DATA_BLOCK "dbtags_Sterowanie"   // DB1
{ S7_Optimized_Access := 'FALSE' }
VERSION : 0.1
// stored: AutoNumber false, DBAccessibleFromOPCUA true, IsOnlyStoredInLoadMemory false, IsWriteProtectedInAS false
   VAR RETAIN
      PID_Compact : Struct
         Setpoint : Real := 1.5;
         Input : Real;
         Input_PER : Int;
         Disturbance : Real;
         ManualEnable : Bool;
         ManualValue : Real;
         ErrorAck : Bool;
         Reset : Bool;
         ModeActivate : Bool;
         Mode : Int := 3;
         ScaledInput : Real;
         Output : Real;
         Output_PER : Int;
         Output_PWM : Bool;
         SetpointLimit_H : Bool;
         SetpointLimit_L : Bool;
         InputWarning_H : Bool;
         InputWarning_L : Bool;
         State : Int;
         Error : Bool;
         ErrorBits : DWord;
      END_STRUCT;
      Tuning : Struct
         Mode : Int := 1;
         Mode_visible : Bool;
         SUT_visible : Bool;
         TIR_visible : Bool;
         last_state : Int;
      END_STRUCT;
      HMI : Struct
         PhysicalUnit : String[5] := '1/min';
         Output_PWM_USInt : USInt;
         "position reached" : Bool;
         ManualMode_visible : Bool;
         Setpoint_limited : Bool;
         ErrorBits_Int : Int;
         ErrorAck_Int : Int;
         Warning_Int : Int;
         ErrorAck_Int_edge : Bool;   // pamięć zbocza reset PID po error
         ErrorAck : Bool;   // reset błędu PID
         Acknowledge_visible : Bool;
      END_STRUCT;
      Speed : Struct
         encoder : Real;
         rpm : Real;
      END_STRUCT;
      SetupControlPompownia : Struct
         SV : Real := 2.0;
         r_Pv_Norm_OUT_2 : Real := 10.0;   // Zakres górny wejścia In_PER_PID
         r_Pv_Norm_OUT_1 : Real := 0.0;   // Zakres dolny wejścia In_PER_PID
         r_Lmn_Hlm : Real := 100.0;   // Ograniczenie górne wartości procesowej [%] MV
         r_Lmn_Llm : Real := 0.0;   // Ograniczenie dolne wartości procesowej [%] MV
         r_Sp_Hlm : Real := 8.0;   // Ograniczenie H zakresu zadawania wartości ciśnienie SV
         r_Sp_Llm : Real := 0.0;   // Ograniczenie L zakresu zadawania wartości ciśnienia SV
         r_Pv_HWrn : Real := 7.8;   // Ostrzeżenie wysoki dla PV
         r_Pv_LWrn : Real := 5.3;   // Ostrzeżenie niski dla PV
         r_Pv_Hlm : Real := 10.0;   // Przetwornik Limit górny
         r_Pv_Llm : Real := 0.0;   // Przetwornik Limit dlolny
         Time_ONK1 : Int := 90;
         Time_ONK2 : Int := 90;
         Time_OFFK1 : Int := 5;
         Time_OFFK2 : Int := 5;
         TimeHz : Int := 30;
         NO4_Cureent : Real;   // Aktualna zawartość amoniaku
         CureentValue_O2_1 : Real;   // Przyrost ciśnienia 1
         CureentValue_O2_2 : Real;   // Przyrost ciścienia 2
         Data_sek1 : Int;   // Licznik sekund dla pomiaru nr1 funkcji Calculation_of_the_increment
         Data_sek2 : Int;   // Licznik sekund dla pomiaru nr2 funkcji Calculation_of_the_increment
         Static_1 : Word;
         Z11_Status : Word;   // Status napędu copia z SCADA
         Z12_Status : Word;   // Status napędu copia z SCADA
         Static_2 : Real;
         Switch_Aut_Rem_Pompy : Bool;   // Bit przełacznika trybu pracy pomp
         tagsdbSwitch_ModelSterowania : Word;   // Wybur model sterowania0- wyłączone, 1- Dosilanie, 2- Przetłączanie, 3- Automat, 4- Ręczne
         barMax_Manual_Hz : Real := 5.0;   // Instancja wartości zadawanej w trybie manual do regulatora PID gdy ciśnienie w rurociągu max
         CurrentMax_Manual_Hz : Real := 5.0;   // Instancja wartości zadawanej w trybie manual do regulatora PID gdy przeciążony falownik
         Statut_Motor : Byte;   // Byte stanu gotowości pomp
         Mem_Res_setCMD_MC_P1 : Bool;   // Znacznik 50 Hz podtrzymanie przełączenia na sieć
         Mem_Res_setCMD_MC_P2 : Bool;   // Znacznik 50 Hz podtrzymanie przełączenia na sieć
         Mem_Res_setCMD_MC_P3 : Bool;   // Znacznik 50 Hz podtrzymanie przełączenia na sieć
         Switch_In_Analog_Mudbas : Bool;   // Bit przełączeania pomiędzy sygnałem bar z wej analog / Modbus
         PV_HWrn_correction : Real;   // Wspóczninik służący wprowadzeniu korekty ostrzeżenia przekroczenia wartości zadanej ciśnienie
         PV_LWrn_correction : Real;   // Wspóczninik służący wprowadzeniu korekty ostrzeżenia zbyt niskia wartości ciśnieniea w stosunku do zadanej
         TimerSet_O2_Up : IEC_TIMER;   // Czas opóżninia podniesienia zadanej wartości ciśnienia
         TimerSet_O2_Down : IEC_TIMER;   // Czas opóżninia obniżenia zadanej wartości ciśnienia
         Pv_Llm_B8 : Real := -1.0;   // Limit dolny przetwornika ciśnienie B8
         Pv_Hlm_B8 : Real := 2.0;   // Limit górny przetwornika ciśnienia B8
         Time_ONK3 : Int;
         Time_OFFK3 : Int := 0;
         Setpoint_Inverter_Pompy { ExternalAccessible := 'False'; ExternalVisible := 'False'; ExternalWritable := 'False'} : Real;   // Wartość zadana Hz odczytane z Modbus
         Frequency_inverter_Pompy { ExternalAccessible := 'False'; ExternalVisible := 'False'; ExternalWritable := 'False'} : Real;   // Aktualne Hz silniku odczytane z Modbus
         MotorCurrent_Inverter_Pompy { ExternalAccessible := 'False'; ExternalVisible := 'False'; ExternalWritable := 'False'} : Real;   // Prąd na silniku zasilanym z falownika odczytane z Modbus
         NormalCurrent_InverterPompy { ExternalAccessible := 'False'; ExternalVisible := 'False'; ExternalWritable := 'False'} : Real;   // Prąd nominalny falownika odczytane z Modbus
         MaxCurrent_Inverter_Pompy { ExternalAccessible := 'False'; ExternalVisible := 'False'; ExternalWritable := 'False'} : Real;   // Prad Max krótkotrwały odczytane z Modbus
         OverTemp_InverterPompy { ExternalAccessible := 'False'; ExternalVisible := 'False'; ExternalWritable := 'False'} : Word;
         OverVolta_InverterPompy { ExternalAccessible := 'False'; ExternalVisible := 'False'; ExternalWritable := 'False'} : Word;
         PIF_Reset : IEC_TIMER;   // impuls resetu regulatora PID 1
         mbAdresABB_Q1 : Word := 1;   // Adres modbus przepływomierz pompownia
         mbAdresPompy : Word := 26;   // Adres modbus falownik
         mbAdresrezerwa_Q2 : Word;   // Adres modbus przepływomierz magistrala - w Stacji Zasuw
         mbAdres_IDslave : Word := 2;   // Adres modbus MT101
         SubPV_K1 : Real := 0.6;   // Wspólczynnik pomniejszenia wyliczanego ciśnienia napotrzeby wyłączenia dodatowej pompy
         SubPV_K2 : Real := 0.45;   // Wspólczynnik pomniejszenia wyliczanego ciśnieia napotrzeby wyłączenia dodatowej pompy
         Setpoint_Inverter_a { ExternalAccessible := 'False'; ExternalVisible := 'False'; ExternalWritable := 'False'} : Real;   // Wartość zadana Hz odczytane z Modbus
         Frequency_inverter_a { ExternalAccessible := 'False'; ExternalVisible := 'False'; ExternalWritable := 'False'} : Real;   // Aktualne Hz silniku odczytane z Modbus
         MotorCurrent_Inverter_a { ExternalAccessible := 'False'; ExternalVisible := 'False'; ExternalWritable := 'False'} : Real;   // Prąd na silniku zasilanym z falownika odczytane z Modbus
         NormalCurrent_Inverter_a { ExternalAccessible := 'False'; ExternalVisible := 'False'; ExternalWritable := 'False'} : Real;   // Prąd nominalny falownika odczytane z Modbus
         MaxCurrent_Inverter_a { ExternalAccessible := 'False'; ExternalVisible := 'False'; ExternalWritable := 'False'} : Real;   // Prad Max krótkotrwały odczytane z Modbus
         OverTemp_InverterPomp { ExternalAccessible := 'False'; ExternalVisible := 'False'; ExternalWritable := 'False'} : Word;
         OverVolta_InverterPomp { ExternalAccessible := 'False'; ExternalVisible := 'False'; ExternalWritable := 'False'} : Word;
         set_barDN500_B5 { ExternalAccessible := 'False'; ExternalVisible := 'False'; ExternalWritable := 'False'} : Real;   // Zadane ciśnienie dosilanie DN500 na czujniku B5
         set_barDN225_B6 { ExternalAccessible := 'False'; ExternalVisible := 'False'; ExternalWritable := 'False'} : Real;   // Zadane ciśnienie przetłacania DN225 na czujniku B6
         MotorCurrent_Inverter_b { ExternalAccessible := 'False'; ExternalVisible := 'False'; ExternalWritable := 'False'} : Real;   // Prąd na silniku zasilanym z falownika odczytane z Modbus
         NormalCurrent_Inverter_b { ExternalAccessible := 'False'; ExternalVisible := 'False'; ExternalWritable := 'False'} : Real;   // Prąd nominalny falownika odczytane z Modbus
         MaxCurrent_Inverter_b { ExternalAccessible := 'False'; ExternalVisible := 'False'; ExternalWritable := 'False'} : Real;   // Prad Max krótkotrwały odczytane z Modbus
         OverTemp_Inverter_b { ExternalAccessible := 'False'; ExternalVisible := 'False'; ExternalWritable := 'False'} : Word;
         OverVolta_Inverter_b { ExternalAccessible := 'False'; ExternalVisible := 'False'; ExternalWritable := 'False'} : Word;
         actOverCurrent_set : Real;   // Zakres ograniczenia prądowego.
         actOverCurrent_set_a : Real := 0.0;   // Zakres ograniczenia prądowego.
         actOverCurrent_set_b : Real := 0.0;   // Zakres ograniczenia prądowego.
         AnalogFrequency_inverter_a { ExternalAccessible := 'False'; ExternalVisible := 'False'; ExternalWritable := 'False'} : Real;   // Aktualne Hz silniku odczytane z Analog
         AnalogFrequency_inverter_b { ExternalAccessible := 'False'; ExternalVisible := 'False'; ExternalWritable := 'False'} : Real := 0.0;   // Aktualne Hz silniku odczytane z Analog
         MaxHour_InverterBlowerWork : Word := 43200;   // Maksymalny czas pracy pracy ciągłej na falowniku dla kompresorów 43200sek = 12h
         TimerSet_Hz_Up_a : IEC_TIMER;
         TimerSet_Hz_Down_a : IEC_TIMER;
         TimerSet_Hz_Up_b : IEC_TIMER;
         TimerSet_Hz_Down_b : IEC_TIMER;
         TimerGen_Hz_Up_a : IEC_TIMER;
         TimerGen_Hz_Down_a : IEC_TIMER;
         TimerGen_Hz_Up_b : IEC_TIMER;
         TimerGen_Hz_Down_b : IEC_TIMER;
         Mem_Res_setCMD_MC_P4 : Bool;   // Znacznik 50 Hz podtrzymanie przełączenia na sieć
         "ABB_1Master.mode" : Byte := 0;
         "rez_2Master.mode" : Byte := 0;
         "Fal_2Master.mode_1" : Byte := 0;
         "Slave_2Master.mode_2" : Byte := 2;
      END_STRUCT;
      "Paramaetry _Zbiorniki" : Struct   // parametry sterowania
         set_poziom_napełniania : Real := 400.0;   // wartość zadana poziomu napełniania
         set_poziom_opróżniania : Real := 30.0;   // wartość zadana poziomu opróżniania
         set_bity_sterowania_napęami_1 : Word;   // bity sterowania napędami
         set_bity_sterowania_napęami_2 : Word;   // bity sterowania napędami
         set_bity_tryb_napędów_1 : Word;   // bity sterowania przełączaniem trybów pracy
         set_bity_tryb_napędów_2 : Word;   // bity sterowania przełączaniem trybów pracy
         rez_alarm_napędów : Word;   // bity kasowania alarmów napędów
         set_strategia_sterowania : Word := 16#0003;   // Sygnały sterowania strategią pompownia - 0= wyłaczone, 1=dosilanie, 2=przetłaczanie,3=automat, 4=ręczne
         set_sterowanie_cyklem : Word;   // Sygnały sterowania cyklem zbiorniki 0-wyłączone, 1=dobowy, 2=tygodniowy, 3=ręczne
         set_położenie_Z10 : Word;   // zadane położenie procentowe Z10
      END_STRUCT;
      Zbiorniki_Godziny : Struct   // godziny cykli pracy
         start_napełnianie : DTL := DTL#1970-01-01-23:55:00;
         Stop_napełnianie : DTL := DTL#1970-01-01-16:00:00;
         Start_przetłaczanie_1 : DTL := DTL#1970-01-01-18:00:00;
         Stop_przetłaczanie_1 : DTL := DTL#1970-01-01-23:55:00;
         Start_dosilanie_1 : DTL := DTL#1970-01-01-18:00:00;
         Stop_dosilanie_1 : DTL := DTL#1970-01-01-23:55:00;
      END_STRUCT;
      Zbiorniki_sondy : Struct   // parametry sond
         "Pv.LIm_Tank1" : Int := 0;   // zakres pomiarowy dolny
         "Pv.HIm_Tank1" : Int := 400;   // zakres pomiarowy górny
         "Pv.LIm_Tank2" : Int := 0;   // zakres pomiarowy dolny
         "Pv.HIm_Tank2" : Int := 400;   // zakres pomiarowy górny
         "Pv.LIm_Tank3" : Int := 0;   // zakres pomiarowy dolny
         "Pv.HIm_Tank3" : Int := 400;   // zakres pomiarowy górny
      END_STRUCT;
      suction_r_Pv_Hlm : Real := 2.0;   // Przetwornik ssania Limit górny
      suction_r_Pv_Llm : Real := -1.0;   // Przetwornik ssania Limit dlolny
   END_VAR
BEGIN
   SetupControlPompownia.PIF_Reset.PT := T#500ms;
   SetupControlPompownia.TimerSet_Hz_Up_a.PT := T#2M;
   SetupControlPompownia.TimerSet_Hz_Down_a.PT := T#2M;
   SetupControlPompownia.TimerSet_Hz_Up_b.PT := T#2M;
   SetupControlPompownia.TimerSet_Hz_Down_b.PT := T#2M;
   SetupControlPompownia.TimerGen_Hz_Up_a.PT := T#100ms;
   SetupControlPompownia.TimerGen_Hz_Down_a.PT := T#100ms;
   SetupControlPompownia.TimerGen_Hz_Up_b.PT := T#100ms;
   SetupControlPompownia.TimerGen_Hz_Down_b.PT := T#100ms;
END_DATA_BLOCK

DATA_BLOCK "hourWork_setData"   // DB30
{ S7_Optimized_Access := 'FALSE' }
VERSION : 0.1
// stored: AutoNumber false, DBAccessibleFromOPCUA true, IsOnlyStoredInLoadMemory false, IsWriteProtectedInAS false
   VAR RETAIN
      Sek_P1 : Int := 1;   // Licznik sekund
      Sek_P2 : Int := 2;   // Licznik sekund
      Sek_P3 : Int := 3;   // Licznik sekund
      Sek_P4 : Int := 3;
      Edge_P1 : Bool;   // Pamięć zbocza
      Edge_P2 : Bool;   // Pamięć zbocza
      Edge_P3 : Bool;   // Pamięć zbocza
      Edge_P4 : Bool := false;
      Sek_a : Int;   // Licznik sekund
      Sek_b : Int;   // Licznik sekund
      Edge_a : Bool;   // Pamięć zbocza
      Edge_b : Bool;   // Pamięć zbocza
      Sum_sek_hur_P1 : Real;   // Licznik sumator godzin i sekund na potrzeby wyznaczania dumchawy do pracy
      Sum_sek_hur_P2 : Real := 0.0;   // Licznik sumator godzin i sekund na potrzeby wyznaczania dumchawy do pracy
      Sum_sek_hur_P3 : Real := 0.0;   // Licznik sumator godzin i sekund na potrzeby wyznaczania dumchawy do pracy
      Sum_sek_hur_P4 : Real := 0.0;
      HourCounterP1 : DWord;   // Counter Work
      HourCounterP2 : DWord;   // Counter Work
      HourCounterP3 : DWord;   // Counter Work
      HourCounterP4 : DWord;
   END_VAR
BEGIN
END_DATA_BLOCK

DATA_BLOCK "dbMasterData"   // DB35
{ S7_Optimized_Access := 'FALSE' }
VERSION : 0.1
// stored: AutoNumber false, DBAccessibleFromOPCUA true, IsOnlyStoredInLoadMemory false, IsWriteProtectedInAS false
   VAR
      ID6_aktualny_przeływu_Adres_33057 { S7_SetPoint := 'True'} : "typeDataABB_real";   // wielkość przepływu / Wartość aktualnego przepływu
      ID6_Licznik_suma_VF_Adres_33063 : "typeDataABB_real";   // licznik objętości VF / Stan licznika objętości dla przepływu w przód VF
      ID6_Licznik_suma_VR_Adres_33065 { S7_SetPoint := 'True'} : "typeDataABB_real";   // licznik objętości VR / Stan licznika objętości dla przepływu w tył VR
      ID6__VD_Adres_6 { S7_SetPoint := 'True'} : "typeDataABB_real";   // Stan bieżącego różnicowego licznika objętości VD
      ID6___GF_Adres_8 { S7_SetPoint := 'True'} : "typeDataABB_real";   // Stan głównego licznika objętości dla przepływu w przód GF
      ID6__GR_Adres_10 { S7_SetPoint := 'True'} : "typeDataABB_real";   // Sta ngłownego licznika objętości dla przepływu w tył GR
      ID6__GD_Adres_12 { S7_SetPoint := 'True'} : "typeDataABB_real";   // Stan głownego licznika różnicowego GD
      ID6__1000 { S7_SetPoint := 'True'} : "typeDataInverter_Word";   // 8-przekrodzony zakres pracy przetwornika, 20-otwarty obwód cewki, 21zwarcie w obwodzie cewki, 26-brak cieczy w czujniku
      data_rez_Wielkość_przeływu_Adres_0 { S7_SetPoint := 'True'} : "typeDataABB_real";   // wielkość przepływu / Wartość aktualnego przepływu
      data_rez_Licznik_objętość_VF_Adres_2 { S7_SetPoint := 'True'} : "typeDataABB_real";   // licznik objętości VF / Stan licznika objętości dla przepływu w przód VF
      data_rez_Licznik_objętość_VR_Adres_4 { S7_SetPoint := 'True'} : "typeDataABB_real";   // licznik objętości VR / Stan licznika objętości dla przepływu w tył VR
      data_rez_Licznik_różnicowy_VD_Adres_6 { S7_SetPoint := 'True'} : "typeDataABB_real";   // licznik różnicy / Stan bieżącego różnicowego licznika objętości VD
      data_rez_Stan_licz_bjętości_GF_Adres_8 { S7_SetPoint := 'True'} : "typeDataABB_real";   // licznik objetosci GF / Stan głównego licznika objętości dla przepływu w przód GF
      data_rez_Stan_licz_bjętości_GR_Adres_10 { S7_SetPoint := 'True'} : "typeDataABB_real";   // licznik objetości GR / Sta ngłownego licznika objętości dla przepływu w tył GR
      data_rez_Stan_licz_rózicowego_obj_GD_Adres_12 { S7_SetPoint := 'True'} : "typeDataABB_real";   // licznik róznicowy / Stan głownego licznika różnicowego GD
      data_rez_Stan_urządzenia_1000 { S7_SetPoint := 'True'} : "typeDataInverter_Word";   // stan urządzenia / 8-przekrodzony zakres pracy przetwornika, 20-otwarty obwód cewki, 21zwarcie w obwodzie cewki, 26-brak cieczy w czujniku
      ID26_Inver_Control_word_416000_Fal { S7_SetPoint := 'True'} : "typeDataInverter_Word";   // Sowo komtrolneCTW falownika [Uint16, index 0]
      ID26_Inver_setpoint_ref_416020_Fal { S7_SetPoint := 'True'} : "typeDataInverter_Word";   // Słowo wartość zadana Hz [Int16, index -1]
      ID26_Inver_Status_word_416030_Fal { S7_SetPoint := 'True'} : "typeDataInverter_Word";   // Słowo statusu STW falownika [Uint16, index 0]
      ID26_Inver_Frequency_416130_Fal { S7_SetPoint := 'True'} : "typeDataInverter_Word";   // Słowo częstotliwość na wyjściu [Uint16, index -1]
      ID26_Inver_MotorCurrent_416140_Fal { S7_SetPoint := 'True'} : "typeDataInverter_Word";   // Słowo częstotliwość na wyjściu [Uint16, index -2]
      ID26_Inver_DC_Voltage_416300_Fal { S7_SetPoint := 'True'} : "typeDataInverter_Word";   // Słowo napięcia DC na szynie [Uint16, index 0]
      ID26_Inver_Temp_416340_Fal { S7_SetPoint := 'True'} : "typeDataInverter_Word";   // Słowo temperatura invertera [Uint8, index 0]
      ID26_Inver_NomCurrent_416360_Fal { S7_SetPoint := 'True'} : "typeDataInverter_Word";   // Słowo nominalna wartośc prądu falonika[Uint16, index -2]
      ID26_Inver_MaxCurrent_416370_Fal { S7_SetPoint := 'True'} : "typeDataInverter_Word";   // Słowo max prąd falownika [Uint16, index -2]
      ID26_Inver_InDigit_416600_Fal { S7_SetPoint := 'True'} : "typeDataInverter_Word";   // Słowo mampa wejść 18,19,27,33 [Uint16, index -0]
      ID26_Inver_HourWork_415010_Fal { S7_SetPoint := 'True'} : "typeDataInverter_DWord";   // Podwójne słowo czasu pracy falownika [Int32, index -0]
      ID26_Inver_OverTemp_415040_Fal { S7_SetPoint := 'True'} : "typeDataInverter_Word";   // Sowo statusu przekroczenie temperatury[Uint16, index 0]
      ID26_Inver_OverVolts_415050_Fal { S7_SetPoint := 'True'} : "typeDataInverter_Word";   // Sowo statusu przekroczenie napięcia[Uint16, index 0]
      data_RTU_value_0 { S7_SetPoint := 'True'} : "typeDataABB_real";   // Wartość 0.0 pomocnicza wyświetlana podczas błędu pomiaru
   END_VAR
BEGIN
   data_RTU_value_0.data[0] := 0.0;
END_DATA_BLOCK

DATA_BLOCK "dbModbusRTU_Reg"   // DB37
TITLE = Modbus RTU Data
{ S7_Optimized_Access := 'FALSE' }
AUTHOR : RTecmer
VERSION : 0.1
// Dane pomiarowe przekazane z bloku danych master modbus RTU
// stored: AutoNumber true, DBAccessibleFromOPCUA true, IsOnlyStoredInLoadMemory false, IsWriteProtectedInAS false
   VAR
      received_6_Wielkość_przeływu_Adres_0 { S7_SetPoint := 'True'} : "typeDataABB_DWord";   // wielkość przepływu
      received_6_Licznik_objętość_VF_Adres_2 { S7_SetPoint := 'True'} : "typeDataABB_DWord";   // licznik objętości VF
      received_6_Licznik_objętość_VR_Adres_4 { S7_SetPoint := 'True'} : "typeDataABB_DWord";   // licznik objętości VR
      received_6_Licznik_różnicowy_VD_Adres_6 { S7_SetPoint := 'True'} : "typeDataABB_DWord";   // licznik różnicy
      receive_6_Stan_licz_bjętości_GF_Adres_8 { S7_SetPoint := 'True'} : "typeDataABB_DWord";   // licznik objetosci GF
      received_6_Stan_licz_bjętości_GR_Adres_10 { S7_SetPoint := 'True'} : "typeDataABB_DWord";   // licznik objetości GR
      received_6_Stan_licz_rózicowego_obj_GD_Adres_12 { S7_SetPoint := 'True'} : "typeDataABB_DWord";   // licznik róznicowy
      received_6_Stan_urządzenia_1000 { S7_SetPoint := 'True'} : "typeDataInverter_Word";   // stan urządzenia
      received_ROL_aktualny_przeływu_Adres_0 { S7_SetPoint := 'True'} : "typeDataABB_DWord";   // wielkość przepływu
      received_ROL_suma_objętość_VF_Adres_2 { S7_SetPoint := 'True'} : "typeDataABB_DWord";   // licznik objętości VF
      received_ROL_suma_objętość_VR_Adres_4 { S7_SetPoint := 'True'} : "typeDataABB_DWord";   // licznik objętości VR
      received_ROL__VD_Adres_6 { S7_SetPoint := 'True'} : "typeDataABB_DWord";   // licznik różnicy
      received_ROL__GF_Adres_8 { S7_SetPoint := 'True'} : "typeDataABB_DWord";   // licznik objetosci GF
      received_ROL__10 { S7_SetPoint := 'True'} : "typeDataABB_DWord";   // licznik objetości GR
      received_ROL__GD_Adres_12 { S7_SetPoint := 'True'} : "typeDataABB_DWord";   // licznik róznicowy
      received_Data_Stan_urządzenia_1000 { S7_SetPoint := 'True'} : "typeDataInverter_Word";   // stan urządzenia
      receivede26_Inver_Control_word_416000 { S7_SetPoint := 'True'} : "typeDataInverter_Word";   // Sowo komtrolneCTW falownika [Uint16, index 0]
      received26_Inver_setpoint_ref_416020 { S7_SetPoint := 'True'} : "typeDataInverter_Word";   // Słowo wartość zadana Hz [Int16, index -1]
      received26_Inver_Status_word_416030 { S7_SetPoint := 'True'} : "typeDataInverter_Word";   // Słowo statusu STW falownika [Uint16, index 0]
      received26_Inver_Frequency_416130 { S7_SetPoint := 'True'} : "typeDataInverter_Word";   // Słowo częstotliwość na wyjściu [Uint16, index -1]
      received26_Inver_MotorCurrent_416140 { S7_SetPoint := 'True'} : "typeDataInverter_Word";   // Słowo prąd na wyjściu [Uint16, index -2]
      received26_Inver_DC_Voltage_416300 { S7_SetPoint := 'True'} : "typeDataInverter_Word";   // Słowo napięcia DC na szynie [Uint16, index 0]
      received26_Inver_Temp_416340 { S7_SetPoint := 'True'} : "typeDataInverter_Word";   // Słowo temperatura invertera [Uint8, index 0]
      received26_Inver_NomCurrent_416360 { S7_SetPoint := 'True'} : "typeDataInverter_Word";   // Słowo nominalna wartośc prądu falonika[Uint16, index -2]
      received26_Inver_MaxCurrent_416370 { S7_SetPoint := 'True'} : "typeDataInverter_Word";   // Słowo max prąd falownika [Uint16, index -2]
      received26_Inver_InDigit_416600 { S7_SetPoint := 'True'} : "typeDataInverter_Word";   // Słowo mampa wejść 18,19,27,33 [Uint16, index -0]
      received26_Inver_HourWork_415010 { S7_SetPoint := 'True'} : "typeDataInverter_DWord";   // Podwójne słowo czasu pracy falownika [Int32, index -0]
      received26_Inver_OverTemp_415040 { S7_SetPoint := 'True'} : "typeDataInverter_Word";   // Sowo statusu przekroczenie temperatury[Uint16, index 0]
      received26_Inver_OverVolts_415050 { S7_SetPoint := 'True'} : "typeDataInverter_Word";   // Sowo statusu przekroczenie napięcia[Uint16, index 0]
      "Przepływomierz nr1 pompownia" : Struct
         ID6_przeływu_VF_Adres_0 { S7_SetPoint := 'True'} : Real;
         ID6_objętość_VF_Adres_2 { S7_SetPoint := 'True'} : Real;
         "ID6_objętośc RF_Adres_4" { S7_SetPoint := 'True'} : Real;
         ID6_licznik_różnicowy_VD_Adres_6 { S7_SetPoint := 'True'} : Real;
         ID6_licznik_objętości_GF_Adres_8 { S7_SetPoint := 'True'} : Real;
         ID6_Licznik_objętości_GR_Adres_10 { S7_SetPoint := 'True'} : Real;
         ID6_Licznik_różnicowy_GD_Adres_12 { S7_SetPoint := 'True'} : Real;
         ID6_status_przepływomierza_Adres_1000 { S7_SetPoint := 'True'} : Word;
      END_STRUCT;
      "Przepływomierz nr2" : Struct
         received_6_przeływu_VF_Adres_0 { S7_SetPoint := 'True'} : Real;
         received_6_objętość_VF_Adres_2 { S7_SetPoint := 'True'} : Real;
         "received_6_objętośc RF_Adres_4" { S7_SetPoint := 'True'} : Real;
         received_6_licznik_różnicowy_VD_Adres_7 { S7_SetPoint := 'True'} : Real;
         received_6_licznik_objętości_GF_Adres_8 { S7_SetPoint := 'True'} : Real;
         received_6_Licznik_objętości_GR_Adres_10 { S7_SetPoint := 'True'} : Real;
         received_6_Licznik_różnicowy_GD_Adres_12 { S7_SetPoint := 'True'} : Real;
         received_6_status_przepływomierza_Adres_1000 { S7_SetPoint := 'True'} : Word;
      END_STRUCT;
   END_VAR
BEGIN
END_DATA_BLOCK

DATA_BLOCK "dbTags_master_ABB_1"   // DB38
{ S7_Optimized_Access := 'FALSE' }
VERSION : 0.1
// stored: AutoNumber true, DBAccessibleFromOPCUA true, IsOnlyStoredInLoadMemory false, IsWriteProtectedInAS false
   VAR
      "step" : USInt := 1;
      edge : Bool := false;
      modbusCommLoad { S7_SetPoint := 'True'} : "typeModbusCommLoad";
      modbusMaster { S7_SetPoint := 'True'} : "typeModbusMaster";
   END_VAR
BEGIN
END_DATA_BLOCK

DATA_BLOCK "dbTags_master_Fal_1"   // DB74
{ S7_Optimized_Access := 'FALSE' }
VERSION : 0.1
// stored: AutoNumber true, DBAccessibleFromOPCUA true, IsOnlyStoredInLoadMemory false, IsWriteProtectedInAS false
   VAR
      "step" : USInt := 1;
      edge : Bool := false;
      modbusCommLoad { S7_SetPoint := 'True'} : "typeModbusCommLoad";
      modbusMaster { S7_SetPoint := 'True'} : "typeModbusMaster";
   END_VAR
BEGIN
END_DATA_BLOCK

DATA_BLOCK "dbTags_master_MPP04_2"   // DB81
{ S7_Optimized_Access := 'FALSE' }
VERSION : 0.1
// stored: AutoNumber true, DBAccessibleFromOPCUA true, IsOnlyStoredInLoadMemory false, IsWriteProtectedInAS false
   VAR
      "step" : USInt := 1;
      edge : Bool := false;
      modbusCommLoad { S7_SetPoint := 'True'} : "typeModbusCommLoad";
      modbusMaster { S7_SetPoint := 'True'} : "typeModbusMaster";
   END_VAR
BEGIN
END_DATA_BLOCK

DATA_BLOCK "dbTags_master_RTU"   // DB90
TITLE = Master
{ S7_Optimized_Access := 'FALSE' }
AUTHOR : rtecmer
VERSION : 0.1
// Instancja dla funkcji Mdbus RTU komunikacja z masterem MT101
// stored: AutoNumber false, DBAccessibleFromOPCUA true, IsOnlyStoredInLoadMemory false, IsWriteProtectedInAS false
   VAR
      "step" : USInt := 1;
      edge : Bool := false;
      modbusCommLoad { S7_SetPoint := 'True'} : "typeModbusCommLoad";
      modbusMaster { S7_SetPoint := 'True'} : "typeModbusSlave";
   END_VAR
BEGIN
END_DATA_BLOCK

DATA_BLOCK "dbTags_slave_RTU"   // DB79
TITLE = Master
{ S7_Optimized_Access := 'FALSE' }
AUTHOR : rtecmer
VERSION : 0.1
// Instancja dla funkcji Mdbus RTU komunikacja z masterem MT101
// stored: AutoNumber false, DBAccessibleFromOPCUA true, IsOnlyStoredInLoadMemory false, IsWriteProtectedInAS false
   VAR
      "step" : USInt := 1;
      edge : Bool := false;
      modbusCommLoad { S7_SetPoint := 'True'} : "typeModbusCommLoad";
      modbusMaster { S7_SetPoint := 'True'} : "typeModbusSlave";
   END_VAR
BEGIN
END_DATA_BLOCK

DATA_BLOCK "temp_dbHoldRegSlave_to_MT101"   // DB102
{ S7_Optimized_Access := 'FALSE' }
VERSION : 0.1
// stored: AutoNumber false, DBAccessibleFromOPCUA true, IsOnlyStoredInLoadMemory false, IsWriteProtectedInAS false
   VAR
      Status_Sterowanie : Struct
         instPump1 : Int;   // Pompa Status M1
         instPump2 : Int := 0;   // Pompa Status M2
         instPump3 : Int := 0;   // Pompa Status M3
         instPump4 : Int := 0;   // Pompa Status M4
         instvValveZ1 : Int := 0;   // Zasuwa Status Z1
         instvValveZ2 : Int := 0;   // Zasuwa Status Z2
         instvValveZ3 : Int := 0;   // Zasuwa Status Z3
         instvValveZ4 : Int := 0;   // Zasuwa Status Z4
         instvValveZ5 : Int := 0;   // Zasuwa Status Z5
         instvValveZ6 : Int := 0;   // Zasuwa Status Z6
         instvValveZ7 : Int := 0;   // Zasuwa Status Z7
         instvValveZ8 : Int := 0;   // Zasuwa Status Z8
         instvValveZ9 : Int := 0;   // Zasuwa Status Z9
         instvValveZ10 : Int := 0;   // Zasuwa Status Z10
         instvValveZ11 : Int := 0;   // Zasuwa Status Z11
         instvValveZ12 : Int := 0;   // Zasuwa Status Z12
         instControllDrivers_1 : Int := 0;   // Bity sterowania napędami (start, stop, otwórz, zamknij) / Bity sterowania napędami (start, stop, otwórz, zamknij) Pompami M1-M4, Zasuwami Z1, Z2, Z3, Z4
         instControllDrivers_2 : Int := 0;   // Bity przełączenia trybu pracy napędów / Bity sterowania napędami ( otwórz, zamknij, start, stop) Zasuwami Z5, Z6, Z7, Z8, Z9, Z10, Z11, Z12
         instConrol_ManAut_1 : Int := 0;   // Bity przełączenia trybu pracy napędów / Bity przełączenia trybu pracy napędów M1-M4, Zasuwami Z1, Z2, Z3, Z4
         instConrol_ManAut_2 : Int := 0;   // Bity przełączenia trybu pracy napędów / Bity przełączenia trybu pracy napędów Z5, Z6, Z7, Z8, Z9, Z10, Z11, Z12
         instLevelTank1 : Int := 0;   // Poziom zbiornik
         instLevelTank2 : Int := 0;   // Poziom zbiornik
         instLevelTank3 : Int := 0;   // Poziom zbiornik
         instLevelTank4 : Int := 0;   // Poziom zbiornik
         instPosition_Z10 : Int := 0;   // rezerwa / Zadawanie położenia Z10
         instControlClearFault1 : Int := 0;   // Bity kasowania alarmów napędów M1-M4, Z1 - Z12
         instControlSygSter_1 : Int := 0;   // rezerwa / Sygnały sterowania strategią (Bit 53.0 - Wyłączony), (Bit 53.1 - Dosilanie), (Bit 53.2 - Przetłączanie), (Bit 53.3 - Automat), (Bit 53.4 - Ręczne )
         instControlSygSter_2 : Int := 0;   // Sygnały sterowania cyklem (Bit 55.0 - Cykl wyłączony (Bit 55.1 - Cykl dobowy), (Bit 55.2 - Cykl tygodniowy), (Bit 55.3 - Cykl ręczny)
         instCurrent_Inverter : Int := 0;   // Aktualny prądu falownika
         instHz_Inverter : Int := 0;   // Aktualne Hz na falowniku
      END_STRUCT;
      Pomiary : Struct
         instLevelSetfilling : Real;   // Zadany poziom napełniania
         instLevelSetemptying : Real;   // Zadany poziom opróżniania
         instSetbarDN500_B6 : Real;   // Zadany ciśnienie tłóczenia kierunek miasto, Modbus 40035
         instSetbarDN500_B5 : Real;   // Zadana ciśnienie dosilania kierunek dosilanie "0" Modbus 40037
         instSetBarMinB9 : Real;   // Zadawana dolna granica ciśnienia studnia "Granica" Modbus 40039
         instB5bar_act : Real;   // Aktualne ciśnienie zasilania z sieci
         instB6bar_act : Real;   // Aktualne ciśnienie DN225 tłoczny
         instB7bar_act : Real;   // Aktualne ciśnienie DN225 pompy
         instB8bar_act : Real;   // Aktualne ciśnienie ssoncy pomp (zab. Suchobieg)
         instPozitionZ10_act : Real;   // Aktualna pozycja zasuwy Z10
         instFlowDN225_act : Real;   // Przepływ DN225 aktualny MIASTO
         instFlowDN225_sum : Real;   // SUMA przepływu Dolna DN225
         instFlowDN500_act : Real;   // Przepływ DN500 (l/s) aktualny, zasilanie zbiorników, DOSILANIE, Modbus 40055
         instFlowDN500_sum : Real;   // SUMA przepływu Dolna DN500 Modbus 40057
      END_STRUCT;
      Godziny : Struct
         instHourStart_Filling : Int;   // Godzina start napełniania
         instMinutStart_Filling : Int;   // Minuta start napełniania
         instHourStop_Filling : Int;   // Godzina stop napełniania
         instMinutStopt_Filling : Int;   // Minuta stop napełniania
         instHourStart_City : Int;   // Godzina start przetłaczanie miasto DN225
         instMinutStart_City : Int;   // Minuty start przetłaczanie miasto DN225
         instHourStop_City : Int;   // Godzina stop przetłaczanie miasto DN225
         instMinutStopt_City : Int;   // Minuty stop przetłaczanie miasto DN225
         instHourStart_Replen : Int;   // Godzina start przetłaczanie miasto DN225
         instMinutStart_Replen : Int;   // Minuty start przetłaczanie miasto DN225
         instHourStop_Replen : Int;   // Godzina stop przetłaczanie miasto DN225
         instMinutStopt_Replen : Int;   // Minuty stop przetłaczanie miasto DN225
      END_STRUCT;
   END_VAR
BEGIN
END_DATA_BLOCK

DATA_BLOCK "DB31_HMI_AreaPointer"   // DB31
{ S7_Optimized_Access := 'FALSE' }
VERSION : 0.1
// stored: AutoNumber false, DBAccessibleFromOPCUA true, IsOnlyStoredInLoadMemory false, IsWriteProtectedInAS false
   VAR
      Coordination : Word;
      DateTime : DTL;
      JobMailbox : Array[0..3] of Word;
      DataRecord : Array[0..4] of Word;
      ProjectID : Word;
      ScreenNumber : Array[0..4] of Word;
      DateTimePLC : Struct
         DateTime : DTL;
         Reserve_01 : Word;
         Reserve_02 : Word;
      END_STRUCT;
      getPLCMode : Int;
      retValueTime : Word;
      cpuSatus : Bool;
   END_VAR
BEGIN
END_DATA_BLOCK

DATA_BLOCK "Dane_ComunicationControlHMI"   // DB29
TITLE = WatchDog HMI-Krata - S7-Krata
{ S7_Optimized_Access := 'FALSE' }
AUTHOR : rtecmer
VERSION : 0.1
// stored: AutoNumber true, DBAccessibleFromOPCUA true, IsOnlyStoredInLoadMemory false, IsWriteProtectedInAS false
   VAR
      Data_czas_loc : DTL;   // Zegar dla panelu HMI Krata
      WatchDog_WinCC : Word;   // Zmienna kordynująca kontrolę komunikacji od strony PC WinCC.
      SetFaultComunikation_Zasuwy : Int;   // Kontrola komunikacji z HMI
      Data_czas_sys : DTL;   // Zegar dla panelu HMI Krata
      Data_czasHMI : DTL;   // Zegar czytany z funkcji RTC (FC44) zapas
      tempCoordinationHMIRS5 : Int;   // Kontrola CoorditionHMI KDN
      tempWatchDog_WinCC : Word;   // Zmienna kordynująca kontrolę komunikacji od strony PC WinCC.
   END_VAR
BEGIN
END_DATA_BLOCK

DATA_BLOCK "Data_Czas_synch"   // DB32
{ S7_Optimized_Access := 'FALSE' }
VERSION : 0.1
// stored: AutoNumber false, DBAccessibleFromOPCUA true, IsOnlyStoredInLoadMemory false, IsWriteProtectedInAS false
   VAR
      Time_Local_read : DTL;
      Time_System_read : DTL;
      Time_System_write : DTL;
      zegar : Time_Of_Day;
      actTime : Real;
   END_VAR
BEGIN
END_DATA_BLOCK

DATA_BLOCK "DB 333"   // DB333
{ S7_Optimized_Access := 'FALSE' }
AUTHOR : AWP_S7P
FAMILY : WEB
VERSION : 1.0
// stored: AutoNumber false, DBAccessibleFromOPCUA true, IsOnlyStoredInLoadMemory false, IsWriteProtectedInAS false
   VAR
      magic { ExternalAccessible := 'False'; ExternalVisible := 'False'; ExternalWritable := 'False'} : DWord := DW#16#41575043;
      consistency_tag { ExternalAccessible := 'False'; ExternalVisible := 'False'; ExternalWritable := 'False'} : DWord := DW#16#3B3640B8;
      db_version { ExternalAccessible := 'False'; ExternalVisible := 'False'; ExternalWritable := 'False'} : Word := W#16#0001;
      length { ExternalAccessible := 'False'; ExternalVisible := 'False'; ExternalWritable := 'False'} : UInt := 182;
      pagetab_of { ExternalAccessible := 'False'; ExternalVisible := 'False'; ExternalWritable := 'False'} : UInt := 92;
      pagetab_count { ExternalAccessible := 'False'; ExternalVisible := 'False'; ExternalWritable := 'False'} : UInt := 1;
      excludetab_of { ExternalAccessible := 'False'; ExternalVisible := 'False'; ExternalWritable := 'False'} : UInt := 102;
      excludetab_count { ExternalAccessible := 'False'; ExternalVisible := 'False'; ExternalWritable := 'False'} : UInt := 0;
      fragmentlist_of { ExternalAccessible := 'False'; ExternalVisible := 'False'; ExternalWritable := 'False'} : UInt := 102;
      fragmentlist_count { ExternalAccessible := 'False'; ExternalVisible := 'False'; ExternalWritable := 'False'} : UInt := 1;
      fragmenttab_of { ExternalAccessible := 'False'; ExternalVisible := 'False'; ExternalWritable := 'False'} : UInt := 110;
      fragmenttab_count { ExternalAccessible := 'False'; ExternalVisible := 'False'; ExternalWritable := 'False'} : UInt := 1;
      datatab_of { ExternalAccessible := 'False'; ExternalVisible := 'False'; ExternalWritable := 'False'} : UInt := 124;
      datatab_count { ExternalAccessible := 'False'; ExternalVisible := 'False'; ExternalWritable := 'False'} : UInt := 0;
      usenametab_of { ExternalAccessible := 'False'; ExternalVisible := 'False'; ExternalWritable := 'False'} : UInt := 124;
      usenametab_count { ExternalAccessible := 'False'; ExternalVisible := 'False'; ExternalWritable := 'False'} : UInt := 0;
      enumreftab_of { ExternalAccessible := 'False'; ExternalVisible := 'False'; ExternalWritable := 'False'} : UInt := 124;
      enumreftab_count { ExternalAccessible := 'False'; ExternalVisible := 'False'; ExternalWritable := 'False'} : UInt := 0;
      enumtab_of { ExternalAccessible := 'False'; ExternalVisible := 'False'; ExternalWritable := 'False'} : UInt := 124;
      enumtab_count { ExternalAccessible := 'False'; ExternalVisible := 'False'; ExternalWritable := 'False'} : UInt := 0;
      textlist_of { ExternalAccessible := 'False'; ExternalVisible := 'False'; ExternalWritable := 'False'} : UInt := 124;
      textlist_count { ExternalAccessible := 'False'; ExternalVisible := 'False'; ExternalWritable := 'False'} : UInt := 58;
      language_frag_tab_of { ExternalAccessible := 'False'; ExternalVisible := 'False'; ExternalWritable := 'False'} : UInt := 104;
      language_frag_tab_count { ExternalAccessible := 'False'; ExternalVisible := 'False'; ExternalWritable := 'False'} : UInt := 6;
      application_name { ExternalAccessible := 'False'; ExternalVisible := 'False'; ExternalWritable := 'False'} : UInt := 1;
      application_url { ExternalAccessible := 'False'; ExternalVisible := 'False'; ExternalWritable := 'False'} : UInt := 10;
      application_desc { ExternalAccessible := 'False'; ExternalVisible := 'False'; ExternalWritable := 'False'} : UInt := 20;
      enum_defs_fragment_start { ExternalAccessible := 'False'; ExternalVisible := 'False'; ExternalWritable := 'False'} : UInt := 0;
      enum_defs_fragment_count { ExternalAccessible := 'False'; ExternalVisible := 'False'; ExternalWritable := 'False'} : UInt := 0;
      commandstate { ExternalAccessible := 'False'; ExternalVisible := 'False'; ExternalWritable := 'False'} : Struct
         last_error { ExternalAccessible := 'False'; ExternalVisible := 'False'; ExternalWritable := 'False'} : Int := 0;
         debug_mode { ExternalAccessible := 'False'; ExternalVisible := 'False'; ExternalWritable := 'False'} : Int := 0;
         init { ExternalAccessible := 'False'; ExternalVisible := 'False'; ExternalWritable := 'False'} : Bool := True;
         deactivate { ExternalAccessible := 'False'; ExternalVisible := 'False'; ExternalWritable := 'False'} : Bool := False;
         initializing { ExternalAccessible := 'False'; ExternalVisible := 'False'; ExternalWritable := 'False'} : Bool := False;
         error { ExternalAccessible := 'False'; ExternalVisible := 'False'; ExternalWritable := 'False'} : Bool := False;
         deactivating { ExternalAccessible := 'False'; ExternalVisible := 'False'; ExternalWritable := 'False'} : Bool := False;
         deactivated { ExternalAccessible := 'False'; ExternalVisible := 'False'; ExternalWritable := 'False'} : Bool := False;
         initialized { ExternalAccessible := 'False'; ExternalVisible := 'False'; ExternalWritable := 'False'} : Bool := False;
         reserved1 { ExternalAccessible := 'False'; ExternalVisible := 'False'; ExternalWritable := 'False'} : Bool := False;
         reserved2 { ExternalAccessible := 'False'; ExternalVisible := 'False'; ExternalWritable := 'False'} : Byte := B#16#00;
      END_STRUCT;
      requesttab { ExternalAccessible := 'False'; ExternalVisible := 'False'; ExternalWritable := 'False'} : Array[1..4] of Struct
         page_index { ExternalAccessible := 'False'; ExternalVisible := 'False'; ExternalWritable := 'False'} : UInt;
         fragment_index { ExternalAccessible := 'False'; ExternalVisible := 'False'; ExternalWritable := 'False'} : UInt;
         continue { ExternalAccessible := 'False'; ExternalVisible := 'False'; ExternalWritable := 'False'} : Bool;
         "repeat" { ExternalAccessible := 'False'; ExternalVisible := 'False'; ExternalWritable := 'False'} : Bool;
         abort { ExternalAccessible := 'False'; ExternalVisible := 'False'; ExternalWritable := 'False'} : Bool;
         finish { ExternalAccessible := 'False'; ExternalVisible := 'False'; ExternalWritable := 'False'} : Bool;
         idle { ExternalAccessible := 'False'; ExternalVisible := 'False'; ExternalWritable := 'False'} : Bool;
         waiting { ExternalAccessible := 'False'; ExternalVisible := 'False'; ExternalWritable := 'False'} : Bool;
         sending { ExternalAccessible := 'False'; ExternalVisible := 'False'; ExternalWritable := 'False'} : Bool;
         aborting { ExternalAccessible := 'False'; ExternalVisible := 'False'; ExternalWritable := 'False'} : Bool;
         reserved3 { ExternalAccessible := 'False'; ExternalVisible := 'False'; ExternalWritable := 'False'} : Byte;
      END_STRUCT;
      pagetab { ExternalAccessible := 'False'; ExternalVisible := 'False'; ExternalWritable := 'False'} : Array[1..1] of Struct
         index { ExternalAccessible := 'False'; ExternalVisible := 'False'; ExternalWritable := 'False'} : UInt;
         url { ExternalAccessible := 'False'; ExternalVisible := 'False'; ExternalWritable := 'False'} : UInt;
         mime_type { ExternalAccessible := 'False'; ExternalVisible := 'False'; ExternalWritable := 'False'} : UInt;
         fragment_start { ExternalAccessible := 'False'; ExternalVisible := 'False'; ExternalWritable := 'False'} : UInt;
         fragment_num { ExternalAccessible := 'False'; ExternalVisible := 'False'; ExternalWritable := 'False'} : UInt;
      END_STRUCT;
      fragmentlist { ExternalAccessible := 'False'; ExternalVisible := 'False'; ExternalWritable := 'False'} : Array[1..1] of UInt;
      language_frag_tab { ExternalAccessible := 'False'; ExternalVisible := 'False'; ExternalWritable := 'False'} : Struct
         max_language { ExternalAccessible := 'False'; ExternalVisible := 'False'; ExternalWritable := 'False'} : UInt := 0;
         fragment_count { ExternalAccessible := 'False'; ExternalVisible := 'False'; ExternalWritable := 'False'} : UInt := 0;
         nolang_offset { ExternalAccessible := 'False'; ExternalVisible := 'False'; ExternalWritable := 'False'} : UInt := 0;
      END_STRUCT;
      fragmenttab { ExternalAccessible := 'False'; ExternalVisible := 'False'; ExternalWritable := 'False'} : Array[1..1] of Struct
         fragment_name { ExternalAccessible := 'False'; ExternalVisible := 'False'; ExternalWritable := 'False'} : UInt;
         fragment_type { ExternalAccessible := 'False'; ExternalVisible := 'False'; ExternalWritable := 'False'} : Byte;
         fragment_version { ExternalAccessible := 'False'; ExternalVisible := 'False'; ExternalWritable := 'False'} : Byte;
         content_db { ExternalAccessible := 'False'; ExternalVisible := 'False'; ExternalWritable := 'False'} : UInt;
         content_of { ExternalAccessible := 'False'; ExternalVisible := 'False'; ExternalWritable := 'False'} : UInt;
         content_length { ExternalAccessible := 'False'; ExternalVisible := 'False'; ExternalWritable := 'False'} : UInt;
         data_start { ExternalAccessible := 'False'; ExternalVisible := 'False'; ExternalWritable := 'False'} : UInt;
         data_num { ExternalAccessible := 'False'; ExternalVisible := 'False'; ExternalWritable := 'False'} : UInt;
      END_STRUCT;
      textlist { ExternalAccessible := 'False'; ExternalVisible := 'False'; ExternalWritable := 'False'} : Array[1..58] of Byte := 777777446F6C6E6100696E6465782E68746D00777777446F6C6E6100696E6465782E68746D00746578742F68746D6C00696E6465782E68746D00;
   END_VAR
BEGIN
   requesttab[1..4].page_index := 0;
   requesttab[1..4].fragment_index := 0;
   requesttab[1..4].continue := False;
   requesttab[1..4]."repeat" := False;
   requesttab[1..4].abort := False;
   requesttab[1..4].finish := False;
   requesttab[1..4].idle := False;
   requesttab[1..4].waiting := False;
   requesttab[1..4].sending := False;
   requesttab[1..4].aborting := False;
   requesttab[1..4].reserved3 := B#16#00;
   pagetab[1].index := 1;
   pagetab[1].url := 29;
   pagetab[1].mime_type := 39;
   pagetab[1].fragment_start := 1;
   pagetab[1].fragment_num := 1;
   fragmentlist[1] := 1;
   fragmenttab[1].fragment_name := 49;
   fragmenttab[1].fragment_type := B#16#00;
   fragmenttab[1].fragment_version := B#16#00;
   fragmenttab[1].content_db := 334;
   fragmenttab[1].content_of := 0;
   fragmenttab[1].content_length := 0;
   fragmenttab[1].data_start := 0;
   fragmenttab[1].data_num := 0;
END_DATA_BLOCK

DATA_BLOCK "DB 334"   // DB334
{ S7_Optimized_Access := 'FALSE' }
AUTHOR : AWP_S7P
FAMILY : WEB
VERSION : 0.1
// stored: AutoNumber false, DBAccessibleFromOPCUA true, IsOnlyStoredInLoadMemory true, IsWriteProtectedInAS false
   VAR
      MAGIC { ExternalAccessible := 'False'; ExternalVisible := 'False'; ExternalWritable := 'False'} : DWord := DW#16#4157_5046;
      CONSISTENCY_TAG { ExternalAccessible := 'False'; ExternalVisible := 'False'; ExternalWritable := 'False'} : DWord := 993411256;
   END_VAR
BEGIN
END_DATA_BLOCK

DATA_BLOCK "ERR_Enum"   // DB105
{ S7_Optimized_Access := 'TRUE' }
VERSION : 0.1
// stored: AutoNumber false, DBAccessibleFromOPCUA true, IsOnlyStoredInLoadMemory false, IsRetainMemResEnabled false, IsWriteProtectedInAS false, MemoryReserve 0
   VAR
      GetErrorID : Array[0..27] of Word;
      SoftwareError { S7_SetPoint := 'True'} : "stt_ERR_Enum_SoftwareError";
      OB80 : Array[0..5] of Byte;
   END_VAR
BEGIN
   GetErrorID[0] := 16#2503;
   GetErrorID[1] := 16#2520;
   GetErrorID[2] := 16#2522;
   GetErrorID[3] := 16#2523;
   GetErrorID[4] := 16#2524;
   GetErrorID[5] := 16#2525;
   GetErrorID[6] := 16#2528;
   GetErrorID[7] := 16#2529;
   GetErrorID[8] := 16#252C;
   GetErrorID[9] := 16#2530;
   GetErrorID[10] := 16#2533;
   GetErrorID[11] := 16#2538;
   GetErrorID[12] := 16#2539;
   GetErrorID[13] := 16#253A;
   GetErrorID[14] := 16#253C;
   GetErrorID[15] := 16#253D;
   GetErrorID[16] := 16#253E;
   GetErrorID[17] := 16#253F;
   GetErrorID[18] := 16#2550;
   GetErrorID[19] := 16#2551;
   GetErrorID[20] := 16#2575;
   GetErrorID[21] := 16#2576;
   GetErrorID[22] := 16#2577;
   GetErrorID[23] := 16#25A0;
   GetErrorID[24] := 16#25A1;
   GetErrorID[25] := 16#25A2;
   GetErrorID[26] := 16#2942;
   GetErrorID[27] := 16#2943;
END_DATA_BLOCK

DATA_BLOCK "ERR_ErrorBufferFull"   // DB106
{ S7_Optimized_Access := 'TRUE' }
VERSION : 0.1
// stored: AutoNumber false, DBAccessibleFromOPCUA true, IsOnlyStoredInLoadMemory false, IsRetainMemResEnabled false, IsWriteProtectedInAS false, MemoryReserve 0
   VAR
      Error { S7_SetPoint := 'True'} : ErrorStruct;
   END_VAR
   VAR RETAIN
      SoftwareError { S7_SetPoint := 'True'} : Array[0..4] of "stt_ERR_SoftwareError";
      GetError { S7_SetPoint := 'True'} : Array[0..27] of "stt_ERR_GetError";
      CounterDiagStatusUpdate : UInt;
   END_VAR
BEGIN
END_DATA_BLOCK

DATA_BLOCK "ERR_ErrorOB"   // DB107
{ S7_Optimized_Access := 'TRUE' }
VERSION : 0.1
// stored: AutoNumber false, DBAccessibleFromOPCUA true, IsOnlyStoredInLoadMemory false, IsRetainMemResEnabled false, IsWriteProtectedInAS false, MemoryReserve 0
   VAR RETAIN
      OB80 { S7_SetPoint := 'True'} : Array[0..5] of "stt_ERR_OB80";
   END_VAR
BEGIN
END_DATA_BLOCK

DATA_BLOCK "V_ErrorOB"   // DB108
{ S7_Optimized_Access := 'TRUE' }
VERSION : 0.1
// stored: AutoNumber false, DBAccessibleFromOPCUA true, IsOnlyStoredInLoadMemory false, IsRetainMemResEnabled false, IsWriteProtectedInAS false, MemoryReserve 0
   VAR
      StartUp { S7_SetPoint := 'True'} : "stt_ERR_StartUpOB";   // //Error read in OB100
      OB80 : Bool;   // //Executed OB80 Time error interrupt
      ResetErrorOB : Bool;   // //Variable connected with button in web site
   END_VAR
BEGIN
END_DATA_BLOCK

DATA_BLOCK "V_SoftwareError"   // DB109
{ S7_Optimized_Access := 'TRUE' }
VERSION : 0.1
// stored: AutoNumber false, DBAccessibleFromOPCUA true, IsOnlyStoredInLoadMemory false, IsRetainMemResEnabled false, IsWriteProtectedInAS false, MemoryReserve 0
   VAR
      SoftwareFunctions : Bool;   // //Error is appear in called function
      GetErrorFunction : Bool;   // //Function GET_ERROR() return error
      DiagnosticBuffer : Bool;   // //Error is appear in diagnostic buffer
      ResetErrorSoftware : Bool;   // //Variable connected with button in web site
   END_VAR
BEGIN
END_DATA_BLOCK

DATA_BLOCK "V_LED"   // DB110
{ S7_Optimized_Access := 'TRUE' }
VERSION : 0.1
// stored: AutoNumber false, DBAccessibleFromOPCUA true, IsOnlyStoredInLoadMemory false, IsRetainMemResEnabled false, IsWriteProtectedInAS false, MemoryReserve 0
   VAR
      LED : Array[1..6] of Int;   // //Status for each module LED
   END_VAR
BEGIN
END_DATA_BLOCK

ORGANIZATION_BLOCK "OB1"   // OB1, LAD, ProgramCycle
TITLE = Głowny blok
{ S7_Optimized_Access := 'TRUE' }
AUTHOR : RTecmer
VERSION : 0.1
// stored: AutoNumber true, IsIECCheckEnabled false, SetENOAutomatically false
   VAR_INPUT
      Initial_Call : Bool;   // Initial call of this OB
      Remanence : Bool;   // =True, if remanent data are available
   END_VAR
   VAR_TEMP
      tempWatchDog_HMI : Int;
   END_VAR
   VAR_TEMP   // added for the SCL form of the ladder/FBD networks
      _w1 : Bool;
      _w2 : Bool;
   END_VAR
BEGIN

REGION Network 2: Zegart RTC
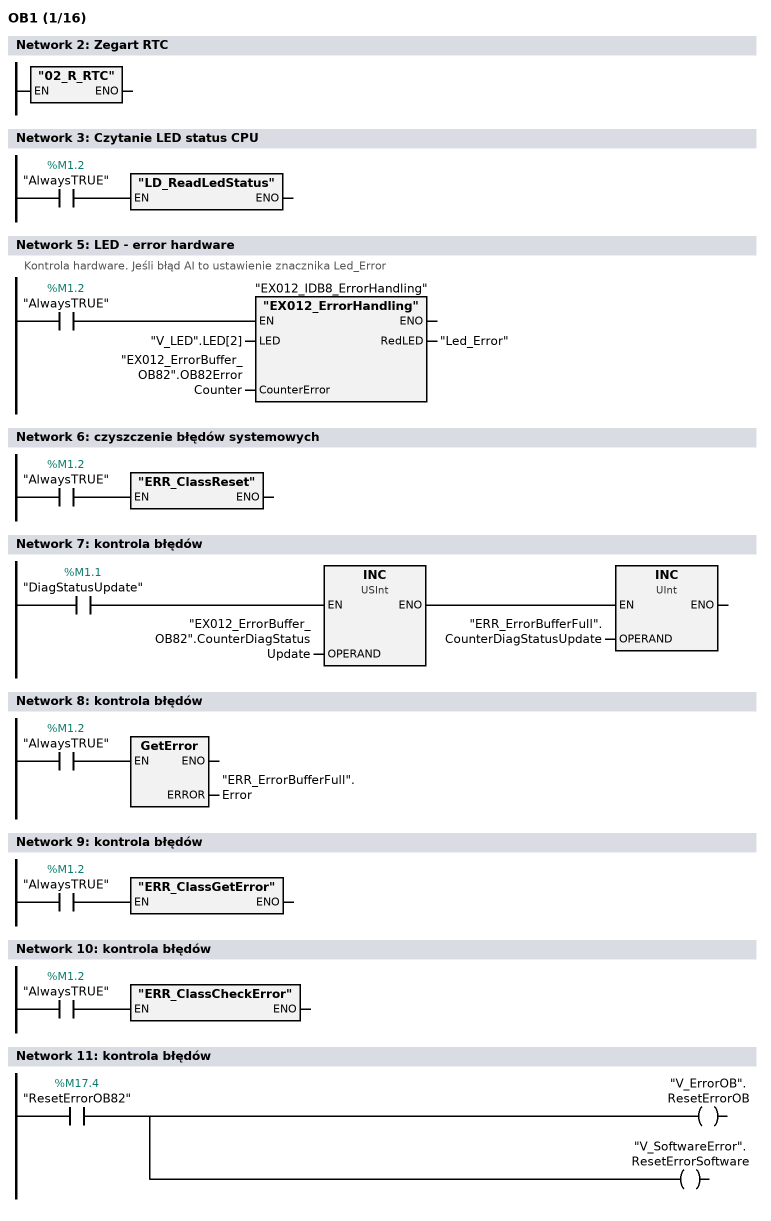
   RUNG wire#powerrail
      "02_R_RTC"()
   END_RUNG
   // the same network as SCL:
   "02_R_RTC"();
END_REGION

REGION Network 3: Czytanie LED status CPU
   RUNG wire#powerrail
      Contact( "AlwaysTRUE" )
      "LD_ReadLedStatus"()
   END_RUNG
   // the same network as SCL:
   IF "AlwaysTRUE" THEN "LD_ReadLedStatus"(); END_IF;
END_REGION

REGION Network 4 (SCL): LED kontrola RUN
   // Przekazanie  stanu LED 1 CPU
   "DB31_HMI_AreaPointer".getPLCMode := "V_LED".LED[1];
END_REGION

REGION Network 5: LED - error hardware
   // Kontrola hardware. Jeśli błąd AI to ustawienie znacznika Led_Error
   RUNG wire#powerrail
      Contact( "AlwaysTRUE" )
      "EX012_IDB8_ErrorHandling"(LED := "V_LED".LED[2], CounterError := "EX012_ErrorBuffer_OB82".OB82ErrorCounter, RedLED => "Led_Error")
   END_RUNG
   // the same network as SCL:
   IF "AlwaysTRUE" THEN
       "EX012_IDB8_ErrorHandling"(LED := "V_LED".LED[2],   // "EX012_ErrorHandling"
                               CounterError := "EX012_ErrorBuffer_OB82".OB82ErrorCounter,
                               RedLED => "Led_Error");
   END_IF;
END_REGION

REGION Network 6: czyszczenie błędów systemowych
   RUNG wire#powerrail
      Contact( "AlwaysTRUE" )
      "ERR_ClassReset"()
   END_RUNG
   // the same network as SCL:
   IF "AlwaysTRUE" THEN "ERR_ClassReset"(); END_IF;
END_REGION

REGION Network 7: kontrola błędów
   RUNG wire#powerrail
      Contact( "DiagStatusUpdate" )
      { S7_Templates := "DestType := USInt" } Inc( "EX012_ErrorBuffer_OB82".CounterDiagStatusUpdate )
      { S7_Templates := "DestType := UInt" } Inc( "ERR_ErrorBufferFull".CounterDiagStatusUpdate )
   END_RUNG
   // the same network as SCL:
   IF "DiagStatusUpdate" THEN
       "EX012_ErrorBuffer_OB82".CounterDiagStatusUpdate := "EX012_ErrorBuffer_OB82".CounterDiagStatusUpdate + 1;
       "ERR_ErrorBufferFull".CounterDiagStatusUpdate := "ERR_ErrorBufferFull".CounterDiagStatusUpdate + 1;
   END_IF;
END_REGION

REGION Network 8: kontrola błędów
   // no SCL statement known for GetError: written as a call
   IF "AlwaysTRUE" THEN GetError(error => "ERR_ErrorBufferFull".Error); END_IF;
END_REGION

REGION Network 9: kontrola błędów
   RUNG wire#powerrail
      Contact( "AlwaysTRUE" )
      "ERR_ClassGetError"()
   END_RUNG
   // the same network as SCL:
   IF "AlwaysTRUE" THEN "ERR_ClassGetError"(); END_IF;
END_REGION

REGION Network 10: kontrola błędów
   RUNG wire#powerrail
      Contact( "AlwaysTRUE" )
      "ERR_ClassCheckError"()
   END_RUNG
   // the same network as SCL:
   IF "AlwaysTRUE" THEN "ERR_ClassCheckError"(); END_IF;
END_REGION

REGION Network 11: kontrola błędów
   RUNG wire#powerrail
      Contact( "ResetErrorOB82" )
      wire#w1
      Coil( "V_ErrorOB".ResetErrorOB )
   END_RUNG
   RUNG wire#w1
      Coil( "V_SoftwareError".ResetErrorSoftware )
   END_RUNG
   // the same network as SCL:
   "V_ErrorOB".ResetErrorOB := "ResetErrorOB82";
   "V_SoftwareError".ResetErrorSoftware := "ResetErrorOB82";
END_REGION

REGION Network 12: Kasowanie alarmów napędów z poziomu SCADA
   // Komunikacja Modbus RTU - MT101
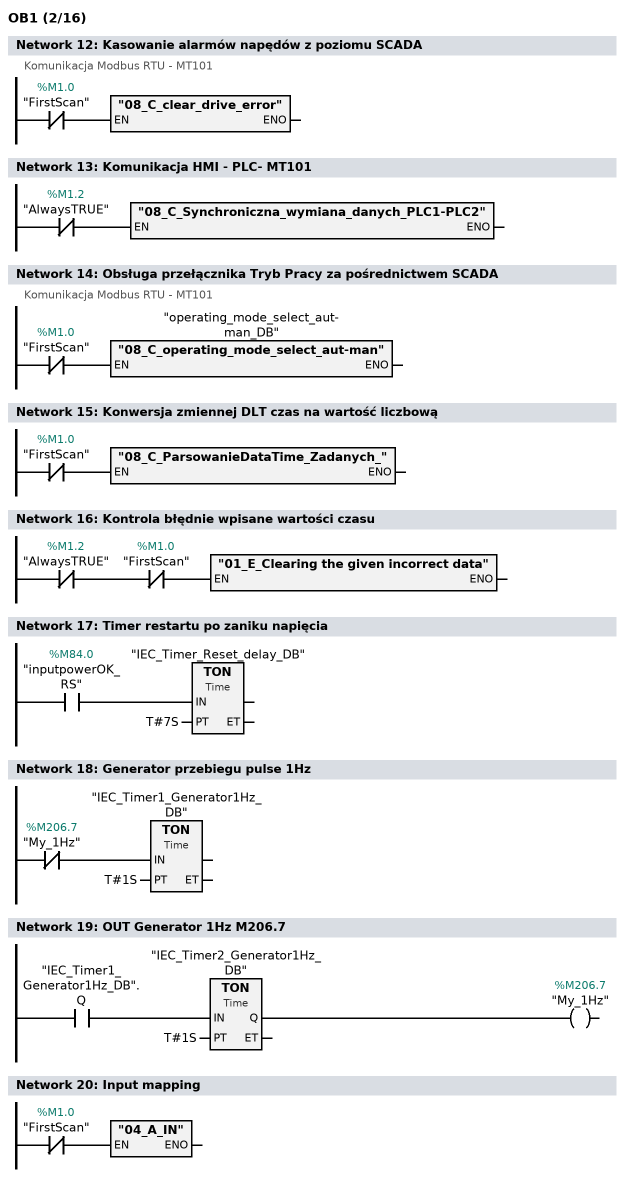
   RUNG wire#powerrail
      I_Contact( "FirstScan" )
      "08_C_clear_drive_error"()
   END_RUNG
   // the same network as SCL:
   IF NOT "FirstScan" THEN "08_C_clear_drive_error"(); END_IF;
END_REGION

REGION Network 13: Komunikacja HMI - PLC- MT101
   RUNG wire#powerrail
      I_Contact( "AlwaysTRUE" )
      "08_C_Synchroniczna_wymiana_danych_PLC1-PLC2"()
   END_RUNG
   // the same network as SCL:
   IF NOT "AlwaysTRUE" THEN "08_C_Synchroniczna_wymiana_danych_PLC1-PLC2"(); END_IF;
END_REGION

REGION Network 14: Obsługa przełącznika Tryb Pracy za pośrednictwem SCADA
   // Komunikacja Modbus RTU - MT101
   RUNG wire#powerrail
      I_Contact( "FirstScan" )
      "operating_mode_select_aut-man_DB"()
   END_RUNG
   // the same network as SCL:
   IF NOT "FirstScan" THEN
       "operating_mode_select_aut-man_DB"();   // "08_C_operating_mode_select_aut-man"
   END_IF;
END_REGION

REGION Network 15: Konwersja zmiennej DLT czas na wartość liczbową
   RUNG wire#powerrail
      I_Contact( "FirstScan" )
      "08_C_ParsowanieDataTime_Zadanych_"()
   END_RUNG
   // the same network as SCL:
   IF NOT "FirstScan" THEN "08_C_ParsowanieDataTime_Zadanych_"(); END_IF;
END_REGION

REGION Network 16: Kontrola błędnie wpisane wartości czasu
   RUNG wire#powerrail
      I_Contact( "AlwaysTRUE" )
      I_Contact( "FirstScan" )
      "01_E_Clearing the given incorrect data"()
   END_RUNG
   // the same network as SCL:
   IF NOT "AlwaysTRUE" AND NOT "FirstScan" THEN "01_E_Clearing the given incorrect data"(); END_IF;
END_REGION

REGION Network 17: Timer restartu po zaniku napięcia
   RUNG wire#powerrail
      Contact( "inputpowerOK_RS" )
      { S7_Templates := "time_type := Time" } "IEC_Timer_Reset_delay_DB".TON(pt := T#7S, et =>)
   END_RUNG
   // the same network as SCL:
   "IEC_Timer_Reset_delay_DB".TON(IN := "inputpowerOK_RS", PT := T#7S);
END_REGION

REGION Network 18: Generator przebiegu pulse 1Hz
   RUNG wire#powerrail
      I_Contact( "My_1Hz" )
      { S7_Templates := "time_type := Time" } "IEC_Timer1_Generator1Hz_DB".TON(pt := T#1S, et =>)
   END_RUNG
   // the same network as SCL:
   "IEC_Timer1_Generator1Hz_DB".TON(IN := NOT "My_1Hz", PT := T#1S);
END_REGION

REGION Network 19: OUT Generator 1Hz M206.7
   RUNG wire#powerrail
      Contact( "IEC_Timer1_Generator1Hz_DB".Q )
      { S7_Templates := "time_type := Time" } "IEC_Timer2_Generator1Hz_DB".TON(pt := T#1S, et =>)
      Coil( "My_1Hz" )
   END_RUNG
   // the same network as SCL:
   "IEC_Timer2_Generator1Hz_DB".TON(IN := "IEC_Timer1_Generator1Hz_DB".Q, PT := T#1S);
   "My_1Hz" := "IEC_Timer2_Generator1Hz_DB".Q;
END_REGION

REGION Network 20: Input mapping
   RUNG wire#powerrail
      I_Contact( "FirstScan" )
      "04_A_IN"()
   END_RUNG
   // the same network as SCL:
   IF NOT "FirstScan" THEN "04_A_IN"(); END_IF;
END_REGION

REGION Network 21: Status napędu Z11 Z12
   // kopiowanie statusu z DB10 do znacznika
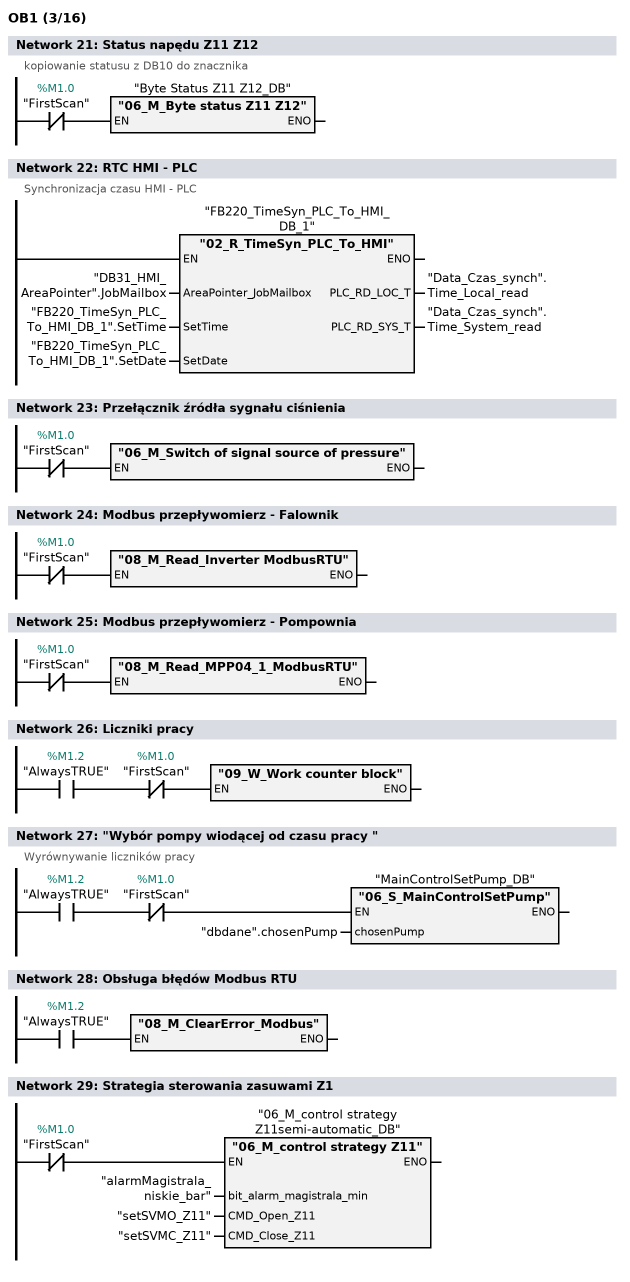
   RUNG wire#powerrail
      I_Contact( "FirstScan" )
      "Byte Status Z11 Z12_DB"()
   END_RUNG
   // the same network as SCL:
   IF NOT "FirstScan" THEN
       "Byte Status Z11 Z12_DB"();   // "06_M_Byte status Z11 Z12"
   END_IF;
END_REGION

REGION Network 22: RTC HMI - PLC
   // Synchronizacja czasu HMI - PLC
   RUNG wire#powerrail
      "FB220_TimeSyn_PLC_To_HMI_DB_1"(AreaPointer_JobMailbox := "DB31_HMI_AreaPointer".JobMailbox, SetTime := "FB220_TimeSyn_PLC_To_HMI_DB_1".SetTime, SetDate := "FB220_TimeSyn_PLC_To_HMI_DB_1".SetDate, PLC_RD_LOC_T => "Data_Czas_synch".Time_Local_read, PLC_RD_SYS_T => "Data_Czas_synch".Time_System_read)
   END_RUNG
   // the same network as SCL:
   "FB220_TimeSyn_PLC_To_HMI_DB_1"(AreaPointer_JobMailbox := "DB31_HMI_AreaPointer".JobMailbox,   // "02_R_TimeSyn_PLC_To_HMI"
                           SetTime := "FB220_TimeSyn_PLC_To_HMI_DB_1".SetTime,
                           SetDate := "FB220_TimeSyn_PLC_To_HMI_DB_1".SetDate,
                           PLC_RD_LOC_T => "Data_Czas_synch".Time_Local_read,
                           PLC_RD_SYS_T => "Data_Czas_synch".Time_System_read);
END_REGION

REGION Network 23: Przełącznik źródła sygnału ciśnienia
   RUNG wire#powerrail
      I_Contact( "FirstScan" )
      "06_M_Switch of signal source of pressure"()
   END_RUNG
   // the same network as SCL:
   IF NOT "FirstScan" THEN "06_M_Switch of signal source of pressure"(); END_IF;
END_REGION

REGION Network 24: Modbus przepływomierz - Falownik
   RUNG wire#powerrail
      I_Contact( "FirstScan" )
      "08_M_Read_Inverter ModbusRTU"()
   END_RUNG
   // the same network as SCL:
   IF NOT "FirstScan" THEN "08_M_Read_Inverter ModbusRTU"(); END_IF;
END_REGION

REGION Network 25: Modbus przepływomierz - Pompownia
   RUNG wire#powerrail
      I_Contact( "FirstScan" )
      "08_M_Read_MPP04_1_ModbusRTU"()
   END_RUNG
   // the same network as SCL:
   IF NOT "FirstScan" THEN "08_M_Read_MPP04_1_ModbusRTU"(); END_IF;
END_REGION

REGION Network 26: Liczniki pracy
   RUNG wire#powerrail
      Contact( "AlwaysTRUE" )
      I_Contact( "FirstScan" )
      "09_W_Work counter block"()
   END_RUNG
   // the same network as SCL:
   IF "AlwaysTRUE" AND NOT "FirstScan" THEN "09_W_Work counter block"(); END_IF;
END_REGION

REGION Network 27: "Wybór pompy wiodącej od czasu pracy "
   // Wyrównywanie liczników pracy
   RUNG wire#powerrail
      Contact( "AlwaysTRUE" )
      I_Contact( "FirstScan" )
      "MainControlSetPump_DB"(chosenPump := "dbdane".chosenPump)
   END_RUNG
   // the same network as SCL:
   IF "AlwaysTRUE" AND NOT "FirstScan" THEN
       "MainControlSetPump_DB"(chosenPump := "dbdane".chosenPump);   // "06_S_MainControlSetPump"
   END_IF;
END_REGION

REGION Network 28: Obsługa błędów Modbus RTU
   RUNG wire#powerrail
      Contact( "AlwaysTRUE" )
      "08_M_ClearError_Modbus"()
   END_RUNG
   // the same network as SCL:
   IF "AlwaysTRUE" THEN "08_M_ClearError_Modbus"(); END_IF;
END_REGION

REGION Network 29: Strategia sterowania zasuwami Z1
   RUNG wire#powerrail
      I_Contact( "FirstScan" )
      "06_M_control strategy Z11semi-automatic_DB"(bit_alarm_magistrala_min := "alarmMagistrala_niskie_bar", CMD_Open_Z11 := "setSVMO_Z11", CMD_Close_Z11 := "setSVMC_Z11")
   END_RUNG
   // the same network as SCL:
   IF NOT "FirstScan" THEN
       "06_M_control strategy Z11semi-automatic_DB"(bit_alarm_magistrala_min := "alarmMagistrala_niskie_bar",   // "06_M_control strategy Z11"
                               CMD_Open_Z11 := "setSVMO_Z11",
                               CMD_Close_Z11 := "setSVMC_Z11");
   END_IF;
END_REGION

REGION Network 30: Alarm max ciśnienie pompownia
   // Wyłaczona od przekroczenie max ciśnienia
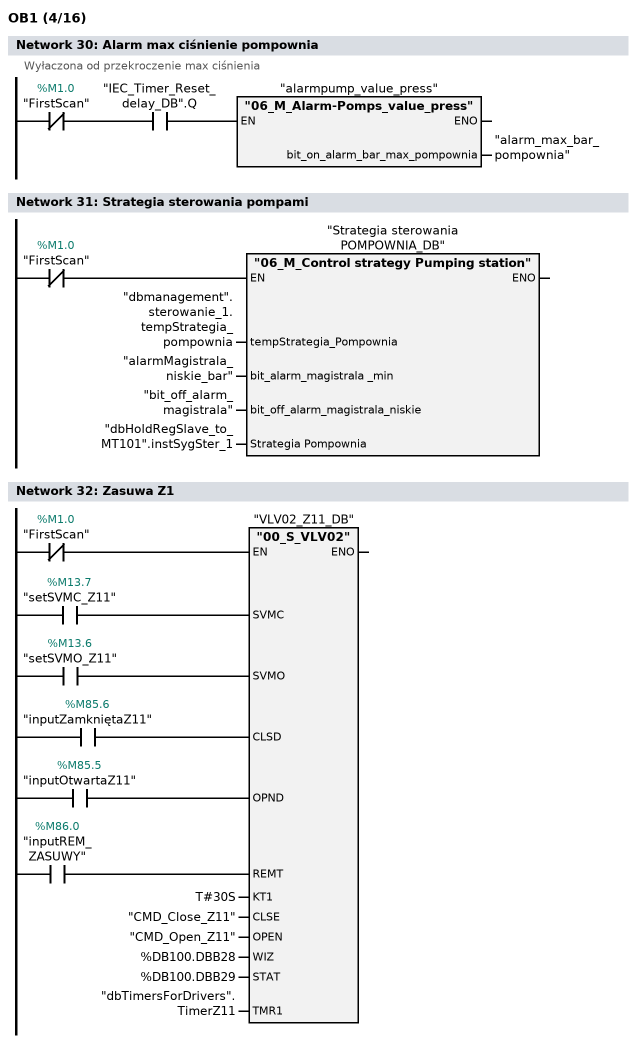
   RUNG wire#powerrail
      I_Contact( "FirstScan" )
      Contact( "IEC_Timer_Reset_delay_DB".Q )
      "alarmpump_value_press"(bit_on_alarm_bar_max_pompownia => "alarm_max_bar_pompownia")
   END_RUNG
   // the same network as SCL:
   IF NOT "FirstScan" AND "IEC_Timer_Reset_delay_DB".Q THEN
       "alarmpump_value_press"(bit_on_alarm_bar_max_pompownia => "alarm_max_bar_pompownia");   // "06_M_Alarm-Pomps_value_press"
   END_IF;
END_REGION

REGION Network 31: Strategia sterowania pompami
   RUNG wire#powerrail
      I_Contact( "FirstScan" )
      "Strategia sterowania POMPOWNIA_DB"(tempStrategia_Pompownia := "dbmanagement".sterowanie_1.tempStrategia_pompownia, "bit_alarm_magistrala _min" := "alarmMagistrala_niskie_bar", bit_off_alarm_magistrala_niskie := "bit_off_alarm_magistrala", "Strategia Pompownia" := "dbHoldRegSlave_to_MT101".instSygSter_1)
   END_RUNG
   // the same network as SCL:
   IF NOT "FirstScan" THEN
       "Strategia sterowania POMPOWNIA_DB"(tempStrategia_Pompownia := "dbmanagement".sterowanie_1.tempStrategia_pompownia,   // "06_M_Control strategy Pumping station"
                               "bit_alarm_magistrala _min" := "alarmMagistrala_niskie_bar",
                               bit_off_alarm_magistrala_niskie := "bit_off_alarm_magistrala",
                               "Strategia Pompownia" := "dbHoldRegSlave_to_MT101".instSygSter_1);
   END_IF;
END_REGION

REGION Network 32: Zasuwa Z1
   RUNG wire#powerrail
      I_Contact( "FirstScan" )
      "VLV02_Z11_DB"(SVMC := wire#w1, SVMO := wire#w2, CLSD := wire#w3, OPND := wire#w4, REMT := wire#w5, KT1 := T#30S, CLSE := "CMD_Close_Z11", OPEN := "CMD_Open_Z11", WIZ := %DB100.DBB28, STAT := %DB100.DBB29, TMR1 := "dbTimersForDrivers".TimerZ11)
   END_RUNG
   RUNG wire#powerrail
      Contact( "setSVMC_Z11" )
   END_RUNG wire#w1
   RUNG wire#powerrail
      Contact( "setSVMO_Z11" )
   END_RUNG wire#w2
   RUNG wire#powerrail
      Contact( "inputZamkniętaZ11" )
   END_RUNG wire#w3
   RUNG wire#powerrail
      Contact( "inputOtwartaZ11" )
   END_RUNG wire#w4
   RUNG wire#powerrail
      Contact( "inputREM_ZASUWY" )
   END_RUNG wire#w5
   // the same network as SCL:
   IF NOT "FirstScan" THEN
       "VLV02_Z11_DB"(SVMC := "setSVMC_Z11",   // "00_S_VLV02"
                      SVMO := "setSVMO_Z11",
                      CLSD := "inputZamkniętaZ11",
                      OPND := "inputOtwartaZ11",
                      REMT := "inputREM_ZASUWY",
                      KT1 := T#30S,
                      CLSE := "CMD_Close_Z11",
                      OPEN := "CMD_Open_Z11",
                      WIZ := %DB100.DBB28,
                      STAT := %DB100.DBB29,
                      TMR1 := "dbTimersForDrivers".TimerZ11);
   END_IF;
END_REGION

REGION Network 33: Konwerter parametrów z falownika
   // funkcja wylicza wartości pobrane z falownika protokołem Modbus RTU
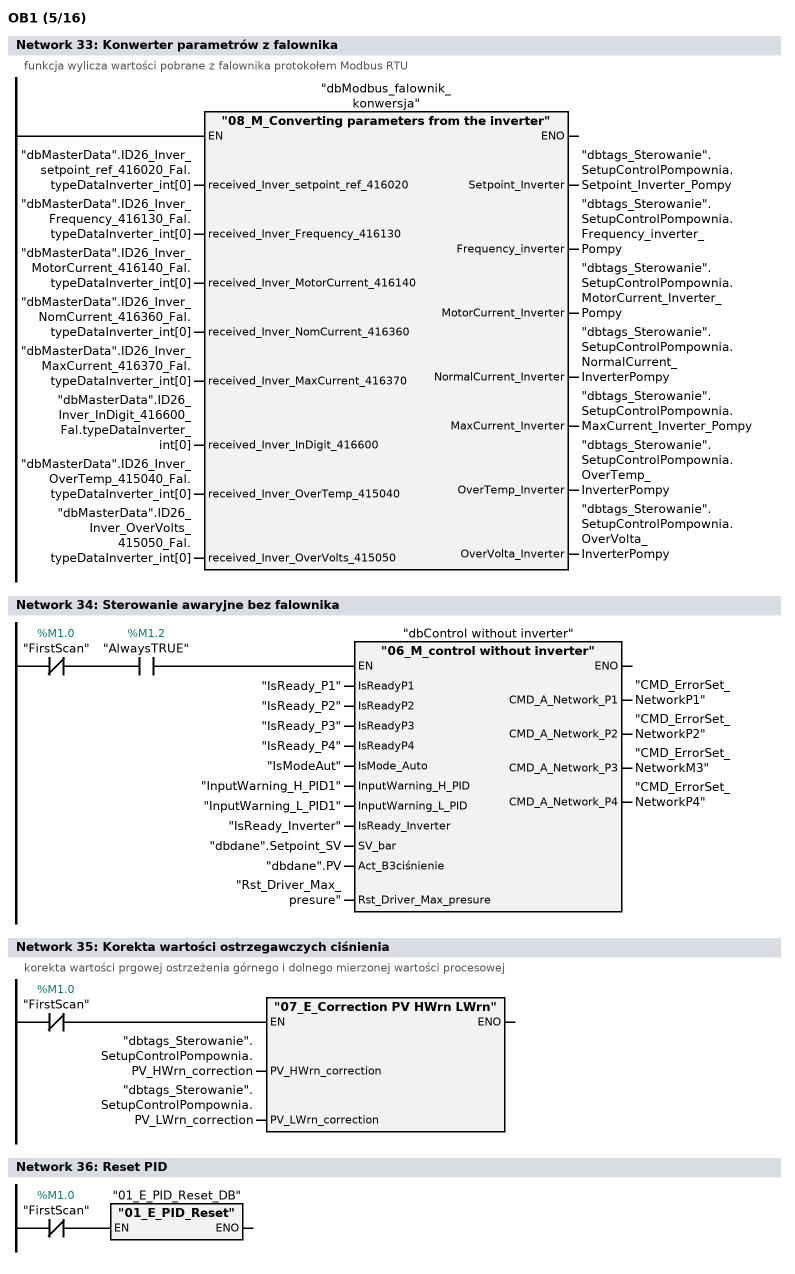
   RUNG wire#powerrail
      "dbModbus_falownik_konwersja"(received_Inver_setpoint_ref_416020 := "dbMasterData".ID26_Inver_setpoint_ref_416020_Fal.typeDataInverter_int[0], received_Inver_Frequency_416130 := "dbMasterData".ID26_Inver_Frequency_416130_Fal.typeDataInverter_int[0], received_Inver_MotorCurrent_416140 := "dbMasterData".ID26_Inver_MotorCurrent_416140_Fal.typeDataInverter_int[0], received_Inver_NomCurrent_416360 := "dbMasterData".ID26_Inver_NomCurrent_416360_Fal.typeDataInverter_int[0], received_Inver_MaxCurrent_416370 := "dbMasterData".ID26_Inver_MaxCurrent_416370_Fal.typeDataInverter_int[0], received_Inver_InDigit_416600 := "dbMasterData".ID26_Inver_InDigit_416600_Fal.typeDataInverter_int[0], received_Inver_OverTemp_415040 := "dbMasterData".ID26_Inver_OverTemp_415040_Fal.typeDataInverter_int[0], received_Inver_OverVolts_415050 := "dbMasterData".ID26_Inver_OverVolts_415050_Fal.typeDataInverter_int[0], Setpoint_Inverter => "dbtags_Sterowanie".SetupControlPompownia.Setpoint_Inverter_Pompy, Frequency_inverter => "dbtags_Sterowanie".SetupControlPompownia.Frequency_inverter_Pompy, MotorCurrent_Inverter => "dbtags_Sterowanie".SetupControlPompownia.MotorCurrent_Inverter_Pompy, NormalCurrent_Inverter => "dbtags_Sterowanie".SetupControlPompownia.NormalCurrent_InverterPompy, MaxCurrent_Inverter => "dbtags_Sterowanie".SetupControlPompownia.MaxCurrent_Inverter_Pompy, OverTemp_Inverter => "dbtags_Sterowanie".SetupControlPompownia.OverTemp_InverterPompy, OverVolta_Inverter => "dbtags_Sterowanie".SetupControlPompownia.OverVolta_InverterPompy)
   END_RUNG
   // the same network as SCL:
   "dbModbus_falownik_konwersja"(received_Inver_setpoint_ref_416020 := "dbMasterData".ID26_Inver_setpoint_ref_416020_Fal.typeDataInverter_int[0],   // "08_M_Converting parameters from the inverter"
                           received_Inver_Frequency_416130 := "dbMasterData".ID26_Inver_Frequency_416130_Fal.typeDataInverter_int[0],
                           received_Inver_MotorCurrent_416140 := "dbMasterData".ID26_Inver_MotorCurrent_416140_Fal.typeDataInverter_int[0],
                           received_Inver_NomCurrent_416360 := "dbMasterData".ID26_Inver_NomCurrent_416360_Fal.typeDataInverter_int[0],
                           received_Inver_MaxCurrent_416370 := "dbMasterData".ID26_Inver_MaxCurrent_416370_Fal.typeDataInverter_int[0],
                           received_Inver_InDigit_416600 := "dbMasterData".ID26_Inver_InDigit_416600_Fal.typeDataInverter_int[0],
                           received_Inver_OverTemp_415040 := "dbMasterData".ID26_Inver_OverTemp_415040_Fal.typeDataInverter_int[0],
                           received_Inver_OverVolts_415050 := "dbMasterData".ID26_Inver_OverVolts_415050_Fal.typeDataInverter_int[0],
                           Setpoint_Inverter => "dbtags_Sterowanie".SetupControlPompownia.Setpoint_Inverter_Pompy,
                           Frequency_inverter => "dbtags_Sterowanie".SetupControlPompownia.Frequency_inverter_Pompy,
                           MotorCurrent_Inverter => "dbtags_Sterowanie".SetupControlPompownia.MotorCurrent_Inverter_Pompy,
                           NormalCurrent_Inverter => "dbtags_Sterowanie".SetupControlPompownia.NormalCurrent_InverterPompy,
                           MaxCurrent_Inverter => "dbtags_Sterowanie".SetupControlPompownia.MaxCurrent_Inverter_Pompy,
                           OverTemp_Inverter => "dbtags_Sterowanie".SetupControlPompownia.OverTemp_InverterPompy,
                           OverVolta_Inverter => "dbtags_Sterowanie".SetupControlPompownia.OverVolta_InverterPompy);
END_REGION

REGION Network 34: Sterowanie awaryjne bez falownika
   RUNG wire#powerrail
      I_Contact( "FirstScan" )
      Contact( "AlwaysTRUE" )
      "dbControl without inverter"(IsReadyP1 := "IsReady_P1", IsReadyP2 := "IsReady_P2", IsReadyP3 := "IsReady_P3", IsReadyP4 := "IsReady_P4", IsMode_Auto := "IsModeAut", InputWarning_H_PID := "InputWarning_H_PID1", InputWarning_L_PID := "InputWarning_L_PID1", IsReady_Inverter := "IsReady_Inverter", SV_bar := "dbdane".Setpoint_SV, Act_B3ciśnienie := "dbdane".PV, Rst_Driver_Max_presure := "Rst_Driver_Max_presure", CMD_A_Network_P1 => "CMD_ErrorSet_NetworkP1", CMD_A_Network_P2 => "CMD_ErrorSet_NetworkP2", CMD_A_Network_P3 => "CMD_ErrorSet_NetworkM3", CMD_A_Network_P4 => "CMD_ErrorSet_NetworkP4")
   END_RUNG
   // the same network as SCL:
   IF NOT "FirstScan" AND "AlwaysTRUE" THEN
       "dbControl without inverter"(IsReadyP1 := "IsReady_P1",   // "06_M_control without inverter"
                               IsReadyP2 := "IsReady_P2",
                               IsReadyP3 := "IsReady_P3",
                               IsReadyP4 := "IsReady_P4",
                               IsMode_Auto := "IsModeAut",
                               InputWarning_H_PID := "InputWarning_H_PID1",
                               InputWarning_L_PID := "InputWarning_L_PID1",
                               IsReady_Inverter := "IsReady_Inverter",
                               SV_bar := "dbdane".Setpoint_SV,
                               Act_B3ciśnienie := "dbdane".PV,
                               Rst_Driver_Max_presure := "Rst_Driver_Max_presure",
                               CMD_A_Network_P1 => "CMD_ErrorSet_NetworkP1",
                               CMD_A_Network_P2 => "CMD_ErrorSet_NetworkP2",
                               CMD_A_Network_P3 => "CMD_ErrorSet_NetworkM3",
                               CMD_A_Network_P4 => "CMD_ErrorSet_NetworkP4");
   END_IF;
END_REGION

REGION Network 35: Korekta wartości ostrzegawczych ciśnienia
   // korekta wartości prgowej ostrzeżenia górnego i dolnego mierzonej wartości procesowej
   RUNG wire#powerrail
      I_Contact( "FirstScan" )
      "07_E_Correction PV HWrn LWrn"(PV_HWrn_correction := "dbtags_Sterowanie".SetupControlPompownia.PV_HWrn_correction, PV_LWrn_correction := "dbtags_Sterowanie".SetupControlPompownia.PV_LWrn_correction)
   END_RUNG
   // the same network as SCL:
   IF NOT "FirstScan" THEN
       "07_E_Correction PV HWrn LWrn"(PV_HWrn_correction := "dbtags_Sterowanie".SetupControlPompownia.PV_HWrn_correction,
                               PV_LWrn_correction := "dbtags_Sterowanie".SetupControlPompownia.PV_LWrn_correction);
   END_IF;
END_REGION

REGION Network 36: Reset PID
   RUNG wire#powerrail
      I_Contact( "FirstScan" )
      "01_E_PID_Reset_DB"()
   END_RUNG
   // the same network as SCL:
   IF NOT "FirstScan" THEN
       "01_E_PID_Reset_DB"();   // "01_E_PID_Reset"
   END_IF;
END_REGION

REGION Network 37: Analog output
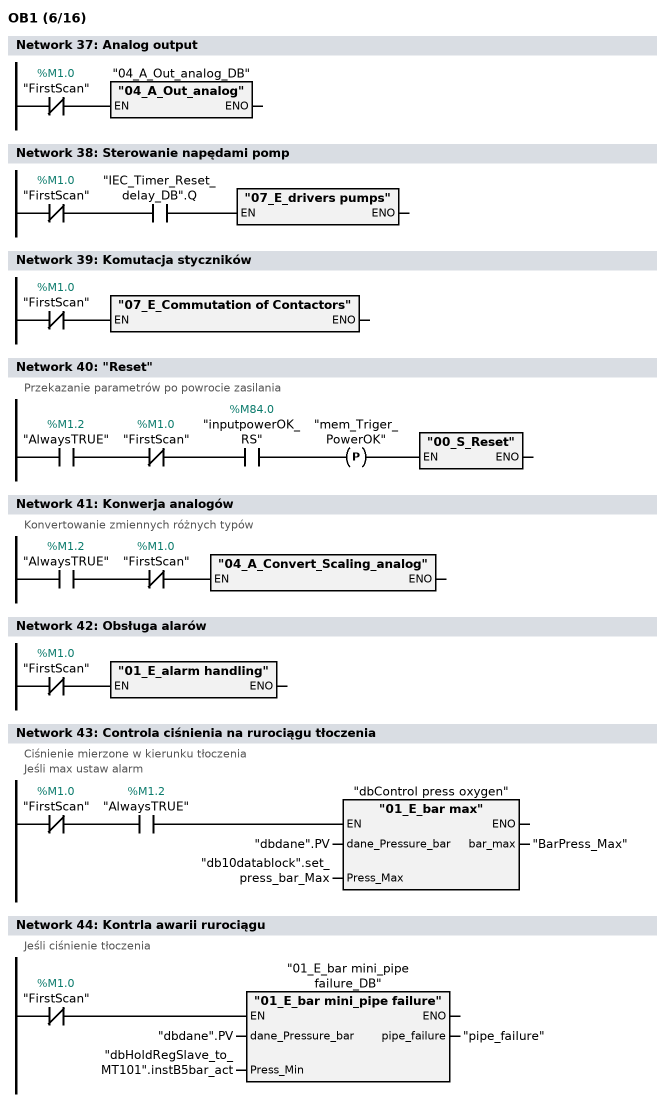
   RUNG wire#powerrail
      I_Contact( "FirstScan" )
      "04_A_Out_analog_DB"()
   END_RUNG
   // the same network as SCL:
   IF NOT "FirstScan" THEN
       "04_A_Out_analog_DB"();   // "04_A_Out_analog"
   END_IF;
END_REGION

REGION Network 38: Sterowanie napędami pomp
   RUNG wire#powerrail
      I_Contact( "FirstScan" )
      Contact( "IEC_Timer_Reset_delay_DB".Q )
      "07_E_drivers pumps"()
   END_RUNG
   // the same network as SCL:
   IF NOT "FirstScan" AND "IEC_Timer_Reset_delay_DB".Q THEN "07_E_drivers pumps"(); END_IF;
END_REGION

REGION Network 39: Komutacja styczników
   RUNG wire#powerrail
      I_Contact( "FirstScan" )
      "07_E_Commutation of Contactors"()
   END_RUNG
   // the same network as SCL:
   IF NOT "FirstScan" THEN "07_E_Commutation of Contactors"(); END_IF;
END_REGION

REGION Network 40: "Reset"
   // Przekazanie parametrów po powrocie zasilania
   RUNG wire#powerrail
      Contact( "AlwaysTRUE" )
      I_Contact( "FirstScan" )
      Contact( "inputpowerOK_RS" )
      P_Trig( "mem_Triger_PowerOK" )
      "00_S_Reset"()
   END_RUNG
   // the same network as SCL:
   #_w1 := "AlwaysTRUE" AND NOT "FirstScan" AND "inputpowerOK_RS";
   #_w2 := #_w1 AND NOT "mem_Triger_PowerOK";   // rising edge
   "mem_Triger_PowerOK" := #_w1;
   IF #_w2 THEN "00_S_Reset"(); END_IF;
END_REGION

REGION Network 41: Konwerja analogów
   // Konvertowanie zmiennych różnych typów
   RUNG wire#powerrail
      Contact( "AlwaysTRUE" )
      I_Contact( "FirstScan" )
      "04_A_Convert_Scaling_analog"()
   END_RUNG
   // the same network as SCL:
   IF "AlwaysTRUE" AND NOT "FirstScan" THEN "04_A_Convert_Scaling_analog"(); END_IF;
END_REGION

REGION Network 42: Obsługa alarów
   RUNG wire#powerrail
      I_Contact( "FirstScan" )
      "01_E_alarm handling"()
   END_RUNG
   // the same network as SCL:
   IF NOT "FirstScan" THEN "01_E_alarm handling"(); END_IF;
END_REGION

REGION Network 43: Controla ciśnienia na rurociągu tłoczenia
   // Ciśnienie mierzone w kierunku tłoczenia
   // Jeśli max ustaw alarm
   RUNG wire#powerrail
      I_Contact( "FirstScan" )
      Contact( "AlwaysTRUE" )
      "dbControl press oxygen"(dane_Pressure_bar := "dbdane".PV, Press_Max := "db10datablock".set_press_bar_Max, bar_max => "BarPress_Max")
   END_RUNG
   // the same network as SCL:
   IF NOT "FirstScan" AND "AlwaysTRUE" THEN
       "dbControl press oxygen"(dane_Pressure_bar := "dbdane".PV,   // "01_E_bar max"
                               Press_Max := "db10datablock".set_press_bar_Max,
                               bar_max => "BarPress_Max");
   END_IF;
END_REGION

REGION Network 44: Kontrla awarii rurociągu
   // Jeśli ciśnienie tłoczenia
   RUNG wire#powerrail
      I_Contact( "FirstScan" )
      "01_E_bar mini_pipe failure_DB"(dane_Pressure_bar := "dbdane".PV, Press_Min := "dbHoldRegSlave_to_MT101".instB5bar_act, pipe_failure => "pipe_failure")
   END_RUNG
   // the same network as SCL:
   IF NOT "FirstScan" THEN
       "01_E_bar mini_pipe failure_DB"(dane_Pressure_bar := "dbdane".PV,   // "01_E_bar mini_pipe failure"
                               Press_Min := "dbHoldRegSlave_to_MT101".instB5bar_act,
                               pipe_failure => "pipe_failure");
   END_IF;
END_REGION

REGION Network 45: Awaryje wyłaczenie pomp dodatkowych od max bar
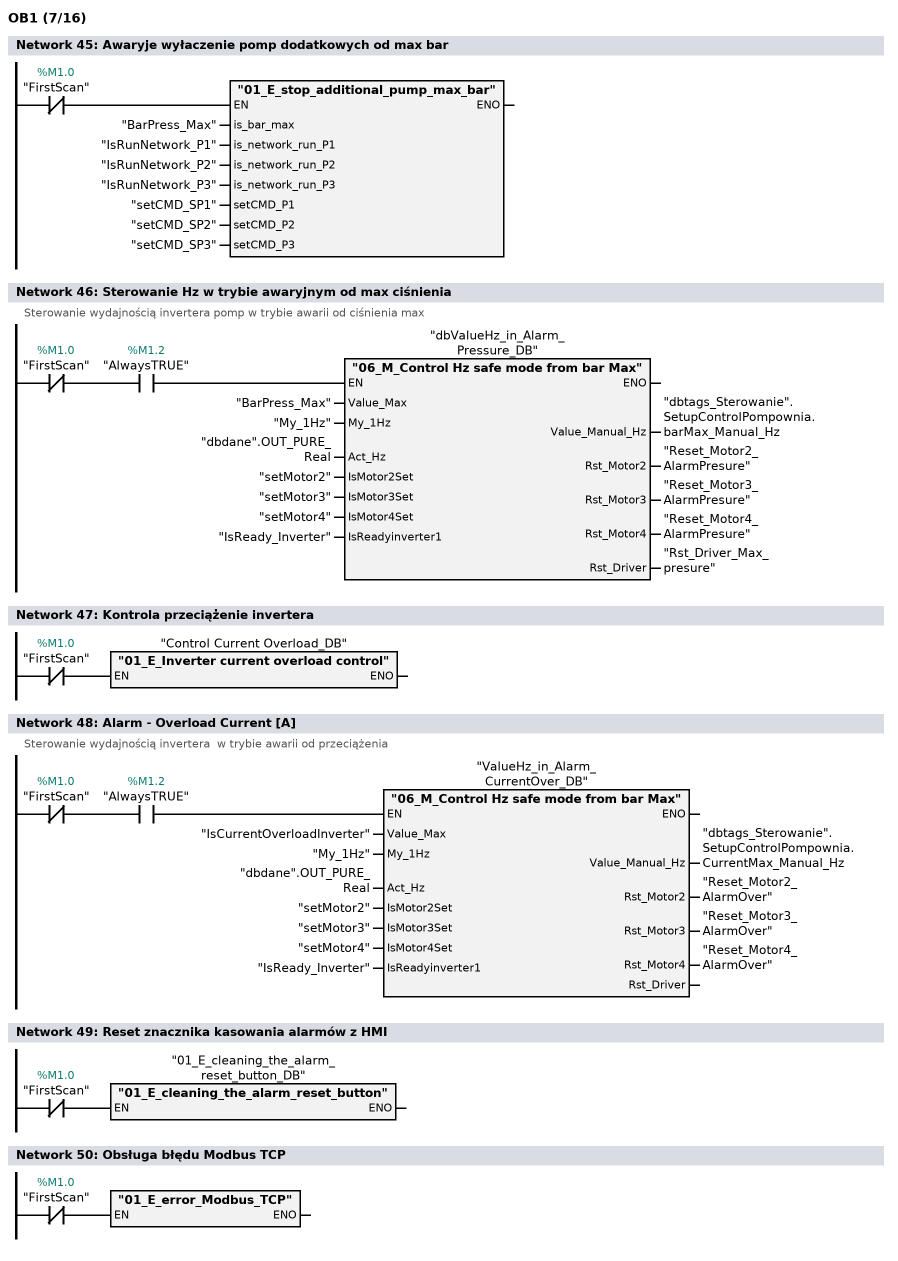
   RUNG wire#powerrail
      I_Contact( "FirstScan" )
      "01_E_stop_additional_pump_max_bar"(is_bar_max := "BarPress_Max", is_network_run_P1 := "IsRunNetwork_P1", is_network_run_P2 := "IsRunNetwork_P2", is_network_run_P3 := "IsRunNetwork_P3", setCMD_P1 := "setCMD_SP1", setCMD_P2 := "setCMD_SP2", setCMD_P3 := "setCMD_SP3")
   END_RUNG
   // the same network as SCL:
   IF NOT "FirstScan" THEN
       "01_E_stop_additional_pump_max_bar"(is_bar_max := "BarPress_Max",
                               is_network_run_P1 := "IsRunNetwork_P1",
                               is_network_run_P2 := "IsRunNetwork_P2",
                               is_network_run_P3 := "IsRunNetwork_P3",
                               setCMD_P1 := "setCMD_SP1",
                               setCMD_P2 := "setCMD_SP2",
                               setCMD_P3 := "setCMD_SP3");
   END_IF;
END_REGION

REGION Network 46: Sterowanie Hz w trybie awaryjnym od max ciśnienia
   // Sterowanie wydajnością invertera pomp w trybie awarii od ciśnienia max
   RUNG wire#powerrail
      I_Contact( "FirstScan" )
      Contact( "AlwaysTRUE" )
      "dbValueHz_in_Alarm_Pressure_DB"(Value_Max := "BarPress_Max", My_1Hz := "My_1Hz", Act_Hz := "dbdane".OUT_PURE_Real, IsMotor2Set := "setMotor2", IsMotor3Set := "setMotor3", IsMotor4Set := "setMotor4", IsReadyinverter1 := "IsReady_Inverter", Value_Manual_Hz => "dbtags_Sterowanie".SetupControlPompownia.barMax_Manual_Hz, Rst_Motor2 => "Reset_Motor2_AlarmPresure", Rst_Motor3 => "Reset_Motor3_AlarmPresure", Rst_Motor4 => "Reset_Motor4_AlarmPresure", Rst_Driver => "Rst_Driver_Max_presure")
   END_RUNG
   // the same network as SCL:
   IF NOT "FirstScan" AND "AlwaysTRUE" THEN
       "dbValueHz_in_Alarm_Pressure_DB"(Value_Max := "BarPress_Max",   // "06_M_Control Hz safe mode from bar Max"
                               My_1Hz := "My_1Hz",
                               Act_Hz := "dbdane".OUT_PURE_Real,
                               IsMotor2Set := "setMotor2",
                               IsMotor3Set := "setMotor3",
                               IsMotor4Set := "setMotor4",
                               IsReadyinverter1 := "IsReady_Inverter",
                               Value_Manual_Hz => "dbtags_Sterowanie".SetupControlPompownia.barMax_Manual_Hz,
                               Rst_Motor2 => "Reset_Motor2_AlarmPresure",
                               Rst_Motor3 => "Reset_Motor3_AlarmPresure",
                               Rst_Motor4 => "Reset_Motor4_AlarmPresure",
                               Rst_Driver => "Rst_Driver_Max_presure");
   END_IF;
END_REGION

REGION Network 47: Kontrola przeciążenie invertera
   RUNG wire#powerrail
      I_Contact( "FirstScan" )
      "Control Current Overload_DB"()
   END_RUNG
   // the same network as SCL:
   IF NOT "FirstScan" THEN
       "Control Current Overload_DB"();   // "01_E_Inverter current overload control"
   END_IF;
END_REGION

REGION Network 48: Alarm - Overload Current [A]
   // Sterowanie wydajnością invertera  w trybie awarii od przeciążenia
   RUNG wire#powerrail
      I_Contact( "FirstScan" )
      Contact( "AlwaysTRUE" )
      "ValueHz_in_Alarm_CurrentOver_DB"(Value_Max := "IsCurrentOverloadInverter", My_1Hz := "My_1Hz", Act_Hz := "dbdane".OUT_PURE_Real, IsMotor2Set := "setMotor2", IsMotor3Set := "setMotor3", IsMotor4Set := "setMotor4", IsReadyinverter1 := "IsReady_Inverter", Value_Manual_Hz => "dbtags_Sterowanie".SetupControlPompownia.CurrentMax_Manual_Hz, Rst_Motor2 => "Reset_Motor2_AlarmOver", Rst_Motor3 => "Reset_Motor3_AlarmOver", Rst_Motor4 => "Reset_Motor4_AlarmOver", Rst_Driver =>)
   END_RUNG
   // the same network as SCL:
   IF NOT "FirstScan" AND "AlwaysTRUE" THEN
       "ValueHz_in_Alarm_CurrentOver_DB"(Value_Max := "IsCurrentOverloadInverter",   // "06_M_Control Hz safe mode from bar Max"
                               My_1Hz := "My_1Hz",
                               Act_Hz := "dbdane".OUT_PURE_Real,
                               IsMotor2Set := "setMotor2",
                               IsMotor3Set := "setMotor3",
                               IsMotor4Set := "setMotor4",
                               IsReadyinverter1 := "IsReady_Inverter",
                               Value_Manual_Hz => "dbtags_Sterowanie".SetupControlPompownia.CurrentMax_Manual_Hz,
                               Rst_Motor2 => "Reset_Motor2_AlarmOver",
                               Rst_Motor3 => "Reset_Motor3_AlarmOver",
                               Rst_Motor4 => "Reset_Motor4_AlarmOver");
   END_IF;
END_REGION

REGION Network 49: Reset znacznika kasowania alarmów z HMI
   RUNG wire#powerrail
      I_Contact( "FirstScan" )
      "01_E_cleaning_the_alarm_reset_button_DB"()
   END_RUNG
   // the same network as SCL:
   IF NOT "FirstScan" THEN
       "01_E_cleaning_the_alarm_reset_button_DB"();   // "01_E_cleaning_the_alarm_reset_button"
   END_IF;
END_REGION

REGION Network 50: Obsługa błędu Modbus TCP
   RUNG wire#powerrail
      I_Contact( "FirstScan" )
      "01_E_error_Modbus_TCP"()
   END_RUNG
   // the same network as SCL:
   IF NOT "FirstScan" THEN "01_E_error_Modbus_TCP"(); END_IF;
END_REGION

REGION Network 51: Konversja Zmiennych
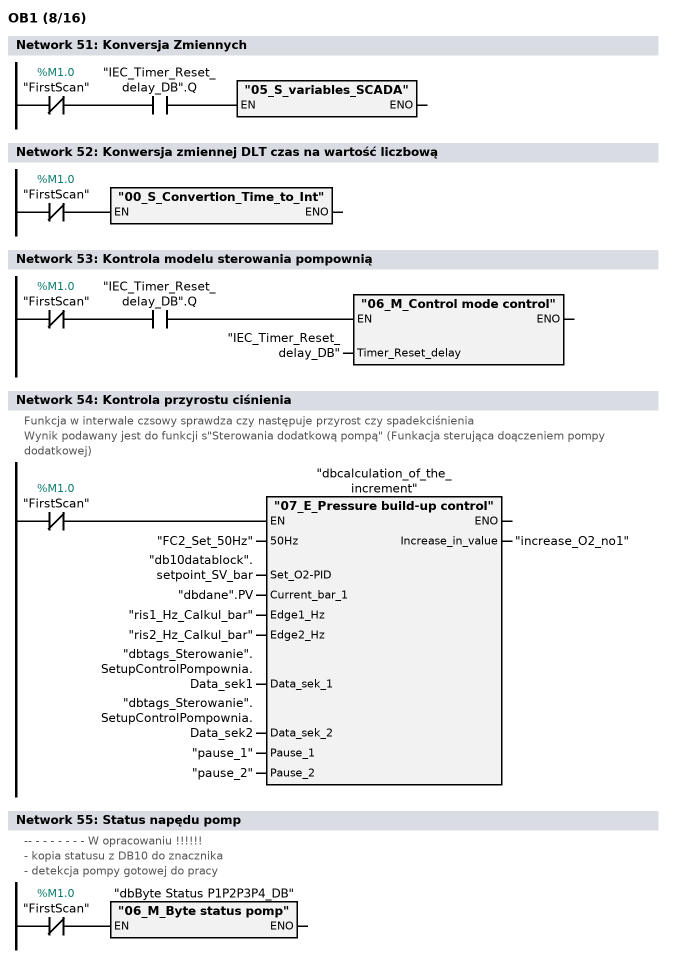
   RUNG wire#powerrail
      I_Contact( "FirstScan" )
      Contact( "IEC_Timer_Reset_delay_DB".Q )
      "05_S_variables_SCADA"()
   END_RUNG
   // the same network as SCL:
   IF NOT "FirstScan" AND "IEC_Timer_Reset_delay_DB".Q THEN "05_S_variables_SCADA"(); END_IF;
END_REGION

REGION Network 52: Konwersja zmiennej DLT czas na wartość liczbową
   RUNG wire#powerrail
      I_Contact( "FirstScan" )
      "00_S_Convertion_Time_to_Int"()
   END_RUNG
   // the same network as SCL:
   IF NOT "FirstScan" THEN "00_S_Convertion_Time_to_Int"(); END_IF;
END_REGION

REGION Network 53: Kontrola modelu sterowania pompownią
   RUNG wire#powerrail
      I_Contact( "FirstScan" )
      Contact( "IEC_Timer_Reset_delay_DB".Q )
      "06_M_Control mode control"(Timer_Reset_delay := "IEC_Timer_Reset_delay_DB")
   END_RUNG
   // the same network as SCL:
   IF NOT "FirstScan" AND "IEC_Timer_Reset_delay_DB".Q THEN
       "06_M_Control mode control"(Timer_Reset_delay := "IEC_Timer_Reset_delay_DB");
   END_IF;
END_REGION

REGION Network 54: Kontrola przyrostu ciśnienia
   // Funkcja w interwale czsowy sprawdza czy następuje przyrost czy spadekciśnienia
   // Wynik podawany jest do funkcji s"Sterowania dodatkową pompą" (Funkacja sterująca doączeniem pompy  dodatkowej)
   RUNG wire#powerrail
      I_Contact( "FirstScan" )
      "dbcalculation_of_the_increment"("50Hz" := "FC2_Set_50Hz", "Set_O2-PID" := "db10datablock".setpoint_SV_bar, Current_bar_1 := "dbdane".PV, Edge1_Hz := "ris1_Hz_Calkul_bar", Edge2_Hz := "ris2_Hz_Calkul_bar", Data_sek_1 := "dbtags_Sterowanie".SetupControlPompownia.Data_sek1, Data_sek_2 := "dbtags_Sterowanie".SetupControlPompownia.Data_sek2, Pause_1 := "pause_1", Pause_2 := "pause_2", Increase_in_value => "increase_O2_no1")
   END_RUNG
   // the same network as SCL:
   IF NOT "FirstScan" THEN
       "dbcalculation_of_the_increment"("50Hz" := "FC2_Set_50Hz",   // "07_E_Pressure build-up control"
                               "Set_O2-PID" := "db10datablock".setpoint_SV_bar,
                               Current_bar_1 := "dbdane".PV,
                               Edge1_Hz := "ris1_Hz_Calkul_bar",
                               Edge2_Hz := "ris2_Hz_Calkul_bar",
                               Data_sek_1 := "dbtags_Sterowanie".SetupControlPompownia.Data_sek1,
                               Data_sek_2 := "dbtags_Sterowanie".SetupControlPompownia.Data_sek2,
                               Pause_1 := "pause_1",
                               Pause_2 := "pause_2",
                               Increase_in_value => "increase_O2_no1");
   END_IF;
END_REGION

REGION Network 55: Status napędu pomp
   // -- - - - - - - - W opracowaniu !!!!!! 
   // - kopia statusu z DB10 do znacznika
   // - detekcja pompy gotowej do pracy
   RUNG wire#powerrail
      I_Contact( "FirstScan" )
      "dbByte Status P1P2P3P4_DB"()
   END_RUNG
   // the same network as SCL:
   IF NOT "FirstScan" THEN
       "dbByte Status P1P2P3P4_DB"();   // "06_M_Byte status pomp"
   END_IF;
END_REGION

REGION Network 56: Sterowanie dołączeniem dodatkowych pomp
   // "dbdane".OUT_PURE_Real
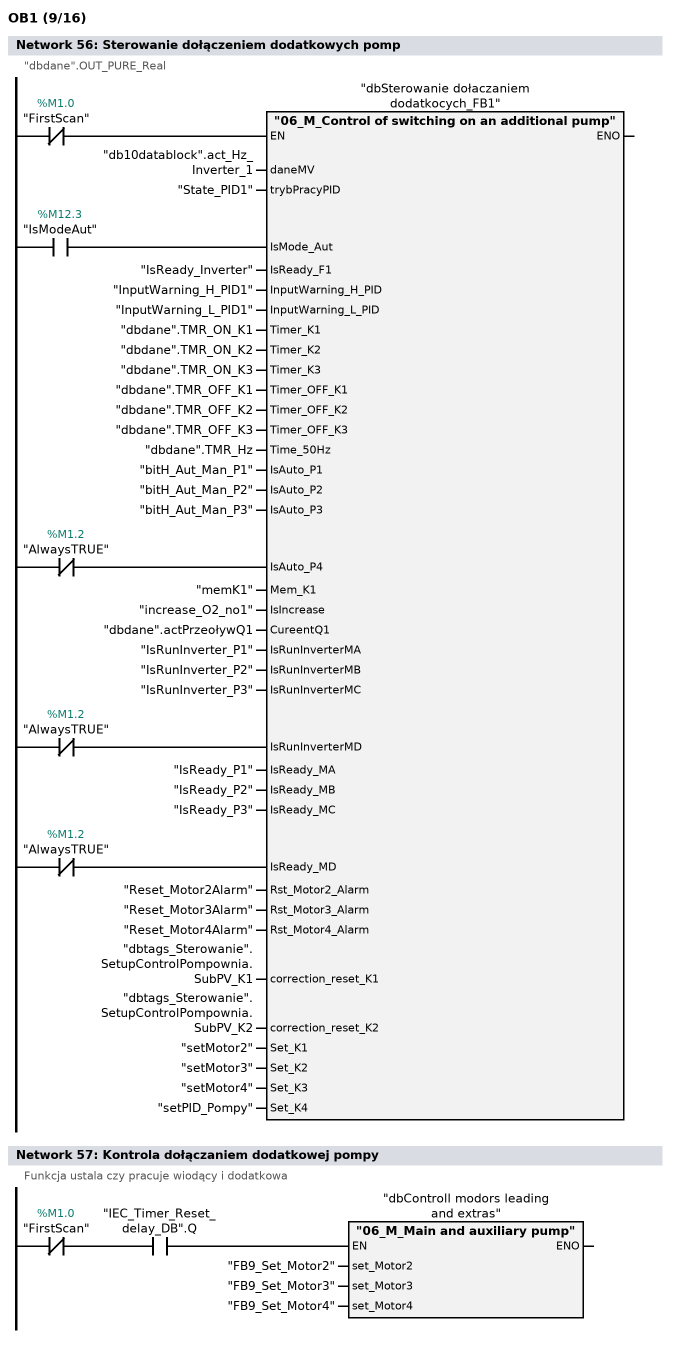
   RUNG wire#powerrail
      I_Contact( "FirstScan" )
      "dbSterowanie dołaczaniem dodatkocych_FB1"(IsMode_Aut := wire#w1, IsAuto_P4 := wire#w2, IsRunInverterMD := wire#w3, IsReady_MD := wire#w4, daneMV := "db10datablock".act_Hz_Inverter_1, trybPracyPID := "State_PID1", IsReady_F1 := "IsReady_Inverter", InputWarning_H_PID := "InputWarning_H_PID1", InputWarning_L_PID := "InputWarning_L_PID1", Timer_K1 := "dbdane".TMR_ON_K1, Timer_K2 := "dbdane".TMR_ON_K2, Timer_K3 := "dbdane".TMR_ON_K3, Timer_OFF_K1 := "dbdane".TMR_OFF_K1, Timer_OFF_K2 := "dbdane".TMR_OFF_K2, Timer_OFF_K3 := "dbdane".TMR_OFF_K3, Time_50Hz := "dbdane".TMR_Hz, IsAuto_P1 := "bitH_Aut_Man_P1", IsAuto_P2 := "bitH_Aut_Man_P2", IsAuto_P3 := "bitH_Aut_Man_P3", Mem_K1 := "memK1", IsIncrease := "increase_O2_no1", CureentQ1 := "dbdane".actPrzeoływQ1, IsRunInverterMA := "IsRunInverter_P1", IsRunInverterMB := "IsRunInverter_P2", IsRunInverterMC := "IsRunInverter_P3", IsReady_MA := "IsReady_P1", IsReady_MB := "IsReady_P2", IsReady_MC := "IsReady_P3", Rst_Motor2_Alarm := "Reset_Motor2Alarm", Rst_Motor3_Alarm := "Reset_Motor3Alarm", Rst_Motor4_Alarm := "Reset_Motor4Alarm", correction_reset_K1 := "dbtags_Sterowanie".SetupControlPompownia.SubPV_K1, correction_reset_K2 := "dbtags_Sterowanie".SetupControlPompownia.SubPV_K2, Set_K1 := "setMotor2", Set_K2 := "setMotor3", Set_K3 := "setMotor4", Set_K4 := "setPID_Pompy")
   END_RUNG
   RUNG wire#powerrail
      Contact( "IsModeAut" )
   END_RUNG wire#w1
   RUNG wire#powerrail
      I_Contact( "AlwaysTRUE" )
   END_RUNG wire#w2
   RUNG wire#powerrail
      I_Contact( "AlwaysTRUE" )
   END_RUNG wire#w3
   RUNG wire#powerrail
      I_Contact( "AlwaysTRUE" )
   END_RUNG wire#w4
   // the same network as SCL:
   IF NOT "FirstScan" THEN
       "dbSterowanie dołaczaniem dodatkocych_FB1"(daneMV := "db10datablock".act_Hz_Inverter_1,   // "06_M_Control of switching on an additional pump"
                               trybPracyPID := "State_PID1",
                               IsMode_Aut := "IsModeAut",
                               IsReady_F1 := "IsReady_Inverter",
                               InputWarning_H_PID := "InputWarning_H_PID1",
                               InputWarning_L_PID := "InputWarning_L_PID1",
                               Timer_K1 := "dbdane".TMR_ON_K1,
                               Timer_K2 := "dbdane".TMR_ON_K2,
                               Timer_K3 := "dbdane".TMR_ON_K3,
                               Timer_OFF_K1 := "dbdane".TMR_OFF_K1,
                               Timer_OFF_K2 := "dbdane".TMR_OFF_K2,
                               Timer_OFF_K3 := "dbdane".TMR_OFF_K3,
                               Time_50Hz := "dbdane".TMR_Hz,
                               IsAuto_P1 := "bitH_Aut_Man_P1",
                               IsAuto_P2 := "bitH_Aut_Man_P2",
                               IsAuto_P3 := "bitH_Aut_Man_P3",
                               IsAuto_P4 := NOT "AlwaysTRUE",
                               Mem_K1 := "memK1",
                               IsIncrease := "increase_O2_no1",
                               CureentQ1 := "dbdane".actPrzeoływQ1,
                               IsRunInverterMA := "IsRunInverter_P1",
                               IsRunInverterMB := "IsRunInverter_P2",
                               IsRunInverterMC := "IsRunInverter_P3",
                               IsRunInverterMD := NOT "AlwaysTRUE",
                               IsReady_MA := "IsReady_P1",
                               IsReady_MB := "IsReady_P2",
                               IsReady_MC := "IsReady_P3",
                               IsReady_MD := NOT "AlwaysTRUE",
                               Rst_Motor2_Alarm := "Reset_Motor2Alarm",
                               Rst_Motor3_Alarm := "Reset_Motor3Alarm",
                               Rst_Motor4_Alarm := "Reset_Motor4Alarm",
                               correction_reset_K1 := "dbtags_Sterowanie".SetupControlPompownia.SubPV_K1,
                               correction_reset_K2 := "dbtags_Sterowanie".SetupControlPompownia.SubPV_K2,
                               Set_K1 := "setMotor2",
                               Set_K2 := "setMotor3",
                               Set_K3 := "setMotor4",
                               Set_K4 := "setPID_Pompy");
   END_IF;
END_REGION

REGION Network 57: Kontrola dołączaniem dodatkowej pompy
   // Funkcja ustala czy pracuje wiodący i dodatkowa
   RUNG wire#powerrail
      I_Contact( "FirstScan" )
      Contact( "IEC_Timer_Reset_delay_DB".Q )
      "dbControll modors leading and extras"(set_Motor2 := "FB9_Set_Motor2", set_Motor3 := "FB9_Set_Motor3", set_Motor4 := "FB9_Set_Motor4")
   END_RUNG
   // the same network as SCL:
   IF NOT "FirstScan" AND "IEC_Timer_Reset_delay_DB".Q THEN
       "dbControll modors leading and extras"(set_Motor2 := "FB9_Set_Motor2",   // "06_M_Main and auxiliary pump"
                               set_Motor3 := "FB9_Set_Motor3",
                               set_Motor4 := "FB9_Set_Motor4");
   END_IF;
END_REGION

REGION Network 58: Wyłączenie pompy wiodącej po 48h
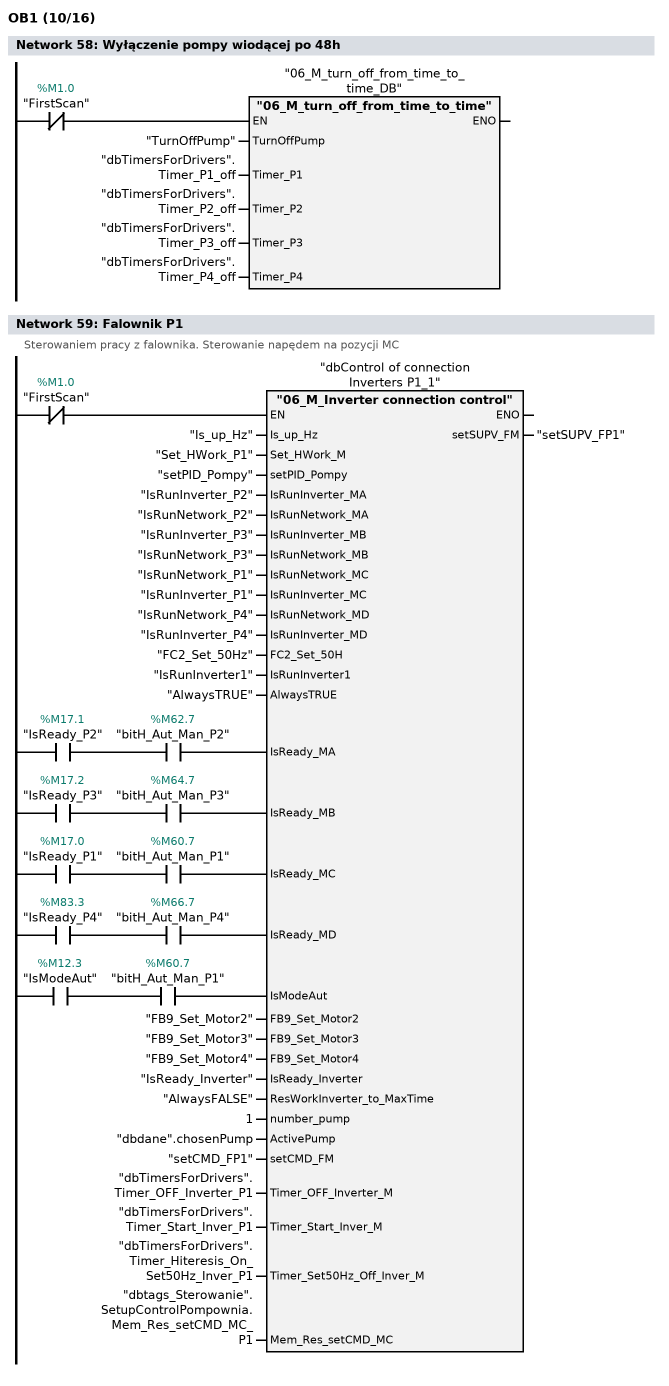
   RUNG wire#powerrail
      I_Contact( "FirstScan" )
      "06_M_turn_off_from_time_to_time_DB"(TurnOffPump := "TurnOffPump", Timer_P1 := "dbTimersForDrivers".Timer_P1_off, Timer_P2 := "dbTimersForDrivers".Timer_P2_off, Timer_P3 := "dbTimersForDrivers".Timer_P3_off, Timer_P4 := "dbTimersForDrivers".Timer_P4_off)
   END_RUNG
   // the same network as SCL:
   IF NOT "FirstScan" THEN
       "06_M_turn_off_from_time_to_time_DB"(TurnOffPump := "TurnOffPump",   // "06_M_turn_off_from_time_to_time"
                               Timer_P1 := "dbTimersForDrivers".Timer_P1_off,
                               Timer_P2 := "dbTimersForDrivers".Timer_P2_off,
                               Timer_P3 := "dbTimersForDrivers".Timer_P3_off,
                               Timer_P4 := "dbTimersForDrivers".Timer_P4_off);
   END_IF;
END_REGION

REGION Network 59: Falownik P1
   // Sterowaniem pracy z falownika. Sterowanie napędem na pozycji MC
   RUNG wire#powerrail
      I_Contact( "FirstScan" )
      "dbControl of connection Inverters P1_1"(IsReady_MA := wire#w1, IsReady_MB := wire#w2, IsReady_MC := wire#w3, IsReady_MD := wire#w4, IsModeAut := wire#w5, Is_up_Hz := "Is_up_Hz", Set_HWork_M := "Set_HWork_P1", setPID_Pompy := "setPID_Pompy", IsRunInverter_MA := "IsRunInverter_P2", IsRunNetwork_MA := "IsRunNetwork_P2", IsRunInverter_MB := "IsRunInverter_P3", IsRunNetwork_MB := "IsRunNetwork_P3", IsRunNetwork_MC := "IsRunNetwork_P1", IsRunInverter_MC := "IsRunInverter_P1", IsRunNetwork_MD := "IsRunNetwork_P4", IsRunInverter_MD := "IsRunInverter_P4", FC2_Set_50H := "FC2_Set_50Hz", IsRunInverter1 := "IsRunInverter1", AlwaysTRUE := "AlwaysTRUE", FB9_Set_Motor2 := "FB9_Set_Motor2", FB9_Set_Motor3 := "FB9_Set_Motor3", FB9_Set_Motor4 := "FB9_Set_Motor4", IsReady_Inverter := "IsReady_Inverter", ResWorkInverter_to_MaxTime := "AlwaysFALSE", number_pump := 1, ActivePump := "dbdane".chosenPump, setCMD_FM := "setCMD_FP1", Timer_OFF_Inverter_M := "dbTimersForDrivers".Timer_OFF_Inverter_P1, Timer_Start_Inver_M := "dbTimersForDrivers".Timer_Start_Inver_P1, Timer_Set50Hz_Off_Inver_M := "dbTimersForDrivers".Timer_Hiteresis_On_Set50Hz_Inver_P1, Mem_Res_setCMD_MC := "dbtags_Sterowanie".SetupControlPompownia.Mem_Res_setCMD_MC_P1, setSUPV_FM => "setSUPV_FP1")
   END_RUNG
   RUNG wire#powerrail
      Contact( "IsReady_P2" )
      Contact( "bitH_Aut_Man_P2" )
   END_RUNG wire#w1
   RUNG wire#powerrail
      Contact( "IsReady_P3" )
      Contact( "bitH_Aut_Man_P3" )
   END_RUNG wire#w2
   RUNG wire#powerrail
      Contact( "IsReady_P1" )
      Contact( "bitH_Aut_Man_P1" )
   END_RUNG wire#w3
   RUNG wire#powerrail
      Contact( "IsReady_P4" )
      Contact( "bitH_Aut_Man_P4" )
   END_RUNG wire#w4
   RUNG wire#powerrail
      Contact( "IsModeAut" )
      Contact( "bitH_Aut_Man_P1" )
   END_RUNG wire#w5
   // the same network as SCL:
   IF NOT "FirstScan" THEN
       "dbControl of connection Inverters P1_1"(Is_up_Hz := "Is_up_Hz",   // "06_M_Inverter connection control"
                               Set_HWork_M := "Set_HWork_P1",
                               setPID_Pompy := "setPID_Pompy",
                               IsRunInverter_MA := "IsRunInverter_P2",
                               IsRunNetwork_MA := "IsRunNetwork_P2",
                               IsRunInverter_MB := "IsRunInverter_P3",
                               IsRunNetwork_MB := "IsRunNetwork_P3",
                               IsRunNetwork_MC := "IsRunNetwork_P1",
                               IsRunInverter_MC := "IsRunInverter_P1",
                               IsRunNetwork_MD := "IsRunNetwork_P4",
                               IsRunInverter_MD := "IsRunInverter_P4",
                               FC2_Set_50H := "FC2_Set_50Hz",
                               IsRunInverter1 := "IsRunInverter1",
                               AlwaysTRUE := "AlwaysTRUE",
                               IsReady_MA := "IsReady_P2" AND "bitH_Aut_Man_P2",
                               IsReady_MB := "IsReady_P3" AND "bitH_Aut_Man_P3",
                               IsReady_MC := "IsReady_P1" AND "bitH_Aut_Man_P1",
                               IsReady_MD := "IsReady_P4" AND "bitH_Aut_Man_P4",
                               IsModeAut := "IsModeAut" AND "bitH_Aut_Man_P1",
                               FB9_Set_Motor2 := "FB9_Set_Motor2",
                               FB9_Set_Motor3 := "FB9_Set_Motor3",
                               FB9_Set_Motor4 := "FB9_Set_Motor4",
                               IsReady_Inverter := "IsReady_Inverter",
                               ResWorkInverter_to_MaxTime := "AlwaysFALSE",
                               number_pump := 1,
                               ActivePump := "dbdane".chosenPump,
                               setCMD_FM := "setCMD_FP1",
                               Timer_OFF_Inverter_M := "dbTimersForDrivers".Timer_OFF_Inverter_P1,
                               Timer_Start_Inver_M := "dbTimersForDrivers".Timer_Start_Inver_P1,
                               Timer_Set50Hz_Off_Inver_M := "dbTimersForDrivers".Timer_Hiteresis_On_Set50Hz_Inver_P1,
                               Mem_Res_setCMD_MC := "dbtags_Sterowanie".SetupControlPompownia.Mem_Res_setCMD_MC_P1,
                               setSUPV_FM => "setSUPV_FP1");
   END_IF;
END_REGION

REGION Network 60: Falownik P2
   // Sterowaniem pracy z falownika. Sterowanie napędem na pozycji MC
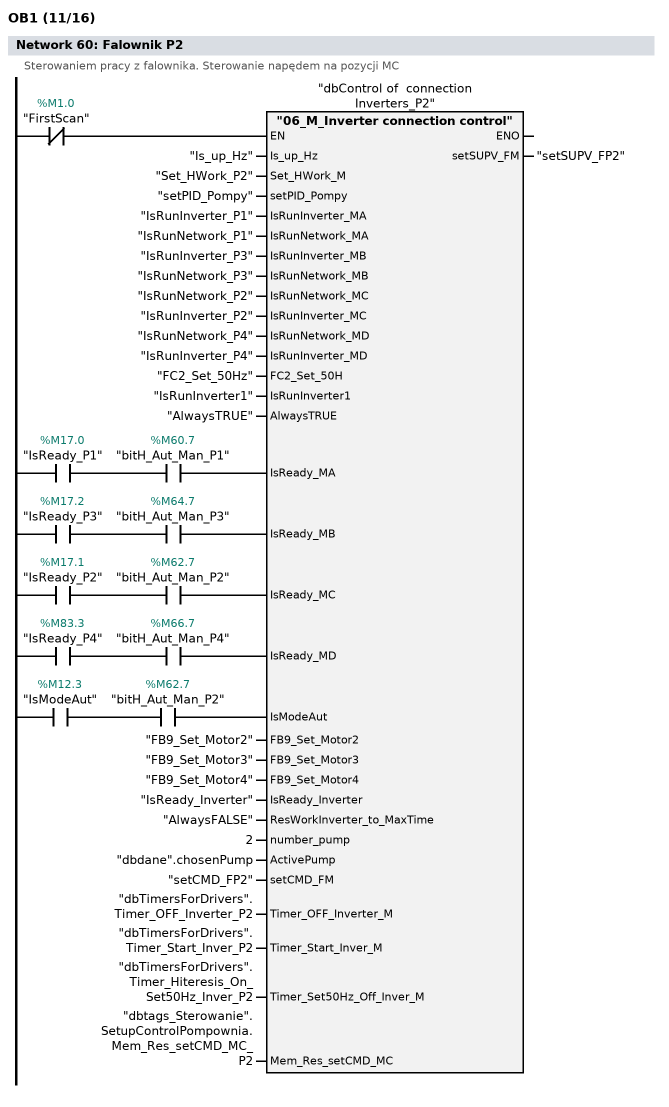
   RUNG wire#powerrail
      I_Contact( "FirstScan" )
      "dbControl of  connection Inverters_P2"(IsReady_MA := wire#w1, IsReady_MB := wire#w2, IsReady_MC := wire#w3, IsReady_MD := wire#w4, IsModeAut := wire#w5, Is_up_Hz := "Is_up_Hz", Set_HWork_M := "Set_HWork_P2", setPID_Pompy := "setPID_Pompy", IsRunInverter_MA := "IsRunInverter_P1", IsRunNetwork_MA := "IsRunNetwork_P1", IsRunInverter_MB := "IsRunInverter_P3", IsRunNetwork_MB := "IsRunNetwork_P3", IsRunNetwork_MC := "IsRunNetwork_P2", IsRunInverter_MC := "IsRunInverter_P2", IsRunNetwork_MD := "IsRunNetwork_P4", IsRunInverter_MD := "IsRunInverter_P4", FC2_Set_50H := "FC2_Set_50Hz", IsRunInverter1 := "IsRunInverter1", AlwaysTRUE := "AlwaysTRUE", FB9_Set_Motor2 := "FB9_Set_Motor2", FB9_Set_Motor3 := "FB9_Set_Motor3", FB9_Set_Motor4 := "FB9_Set_Motor4", IsReady_Inverter := "IsReady_Inverter", ResWorkInverter_to_MaxTime := "AlwaysFALSE", number_pump := 2, ActivePump := "dbdane".chosenPump, setCMD_FM := "setCMD_FP2", Timer_OFF_Inverter_M := "dbTimersForDrivers".Timer_OFF_Inverter_P2, Timer_Start_Inver_M := "dbTimersForDrivers".Timer_Start_Inver_P2, Timer_Set50Hz_Off_Inver_M := "dbTimersForDrivers".Timer_Hiteresis_On_Set50Hz_Inver_P2, Mem_Res_setCMD_MC := "dbtags_Sterowanie".SetupControlPompownia.Mem_Res_setCMD_MC_P2, setSUPV_FM => "setSUPV_FP2")
   END_RUNG
   RUNG wire#powerrail
      Contact( "IsReady_P1" )
      Contact( "bitH_Aut_Man_P1" )
   END_RUNG wire#w1
   RUNG wire#powerrail
      Contact( "IsReady_P3" )
      Contact( "bitH_Aut_Man_P3" )
   END_RUNG wire#w2
   RUNG wire#powerrail
      Contact( "IsReady_P2" )
      Contact( "bitH_Aut_Man_P2" )
   END_RUNG wire#w3
   RUNG wire#powerrail
      Contact( "IsReady_P4" )
      Contact( "bitH_Aut_Man_P4" )
   END_RUNG wire#w4
   RUNG wire#powerrail
      Contact( "IsModeAut" )
      Contact( "bitH_Aut_Man_P2" )
   END_RUNG wire#w5
   // the same network as SCL:
   IF NOT "FirstScan" THEN
       "dbControl of  connection Inverters_P2"(Is_up_Hz := "Is_up_Hz",   // "06_M_Inverter connection control"
                               Set_HWork_M := "Set_HWork_P2",
                               setPID_Pompy := "setPID_Pompy",
                               IsRunInverter_MA := "IsRunInverter_P1",
                               IsRunNetwork_MA := "IsRunNetwork_P1",
                               IsRunInverter_MB := "IsRunInverter_P3",
                               IsRunNetwork_MB := "IsRunNetwork_P3",
                               IsRunNetwork_MC := "IsRunNetwork_P2",
                               IsRunInverter_MC := "IsRunInverter_P2",
                               IsRunNetwork_MD := "IsRunNetwork_P4",
                               IsRunInverter_MD := "IsRunInverter_P4",
                               FC2_Set_50H := "FC2_Set_50Hz",
                               IsRunInverter1 := "IsRunInverter1",
                               AlwaysTRUE := "AlwaysTRUE",
                               IsReady_MA := "IsReady_P1" AND "bitH_Aut_Man_P1",
                               IsReady_MB := "IsReady_P3" AND "bitH_Aut_Man_P3",
                               IsReady_MC := "IsReady_P2" AND "bitH_Aut_Man_P2",
                               IsReady_MD := "IsReady_P4" AND "bitH_Aut_Man_P4",
                               IsModeAut := "IsModeAut" AND "bitH_Aut_Man_P2",
                               FB9_Set_Motor2 := "FB9_Set_Motor2",
                               FB9_Set_Motor3 := "FB9_Set_Motor3",
                               FB9_Set_Motor4 := "FB9_Set_Motor4",
                               IsReady_Inverter := "IsReady_Inverter",
                               ResWorkInverter_to_MaxTime := "AlwaysFALSE",
                               number_pump := 2,
                               ActivePump := "dbdane".chosenPump,
                               setCMD_FM := "setCMD_FP2",
                               Timer_OFF_Inverter_M := "dbTimersForDrivers".Timer_OFF_Inverter_P2,
                               Timer_Start_Inver_M := "dbTimersForDrivers".Timer_Start_Inver_P2,
                               Timer_Set50Hz_Off_Inver_M := "dbTimersForDrivers".Timer_Hiteresis_On_Set50Hz_Inver_P2,
                               Mem_Res_setCMD_MC := "dbtags_Sterowanie".SetupControlPompownia.Mem_Res_setCMD_MC_P2,
                               setSUPV_FM => "setSUPV_FP2");
   END_IF;
END_REGION

REGION Network 61: Falownik P3
   // Sterowaniem pracy z falownika. Sterowanie napędem na pozycji MC
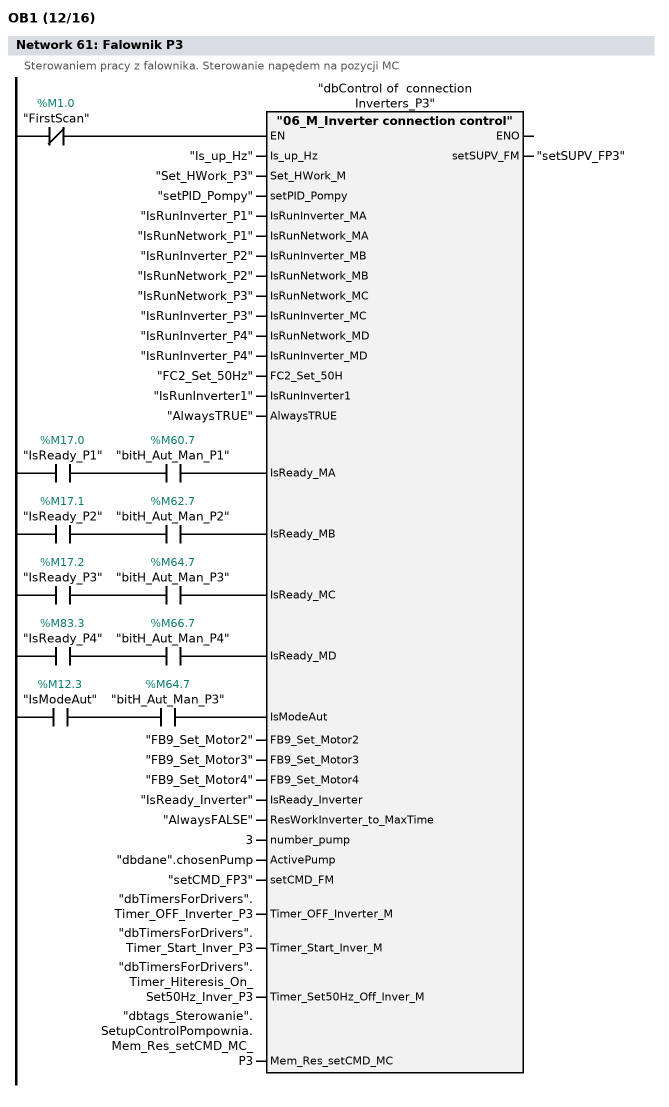
   RUNG wire#powerrail
      I_Contact( "FirstScan" )
      "dbControl of  connection Inverters_P3"(IsReady_MA := wire#w1, IsReady_MB := wire#w2, IsReady_MC := wire#w3, IsReady_MD := wire#w4, IsModeAut := wire#w5, Is_up_Hz := "Is_up_Hz", Set_HWork_M := "Set_HWork_P3", setPID_Pompy := "setPID_Pompy", IsRunInverter_MA := "IsRunInverter_P1", IsRunNetwork_MA := "IsRunNetwork_P1", IsRunInverter_MB := "IsRunInverter_P2", IsRunNetwork_MB := "IsRunNetwork_P2", IsRunNetwork_MC := "IsRunNetwork_P3", IsRunInverter_MC := "IsRunInverter_P3", IsRunNetwork_MD := "IsRunInverter_P4", IsRunInverter_MD := "IsRunInverter_P4", FC2_Set_50H := "FC2_Set_50Hz", IsRunInverter1 := "IsRunInverter1", AlwaysTRUE := "AlwaysTRUE", FB9_Set_Motor2 := "FB9_Set_Motor2", FB9_Set_Motor3 := "FB9_Set_Motor3", FB9_Set_Motor4 := "FB9_Set_Motor4", IsReady_Inverter := "IsReady_Inverter", ResWorkInverter_to_MaxTime := "AlwaysFALSE", number_pump := 3, ActivePump := "dbdane".chosenPump, setCMD_FM := "setCMD_FP3", Timer_OFF_Inverter_M := "dbTimersForDrivers".Timer_OFF_Inverter_P3, Timer_Start_Inver_M := "dbTimersForDrivers".Timer_Start_Inver_P3, Timer_Set50Hz_Off_Inver_M := "dbTimersForDrivers".Timer_Hiteresis_On_Set50Hz_Inver_P3, Mem_Res_setCMD_MC := "dbtags_Sterowanie".SetupControlPompownia.Mem_Res_setCMD_MC_P3, setSUPV_FM => "setSUPV_FP3")
   END_RUNG
   RUNG wire#powerrail
      Contact( "IsReady_P1" )
      Contact( "bitH_Aut_Man_P1" )
   END_RUNG wire#w1
   RUNG wire#powerrail
      Contact( "IsReady_P2" )
      Contact( "bitH_Aut_Man_P2" )
   END_RUNG wire#w2
   RUNG wire#powerrail
      Contact( "IsReady_P3" )
      Contact( "bitH_Aut_Man_P3" )
   END_RUNG wire#w3
   RUNG wire#powerrail
      Contact( "IsReady_P4" )
      Contact( "bitH_Aut_Man_P4" )
   END_RUNG wire#w4
   RUNG wire#powerrail
      Contact( "IsModeAut" )
      Contact( "bitH_Aut_Man_P3" )
   END_RUNG wire#w5
   // the same network as SCL:
   IF NOT "FirstScan" THEN
       "dbControl of  connection Inverters_P3"(Is_up_Hz := "Is_up_Hz",   // "06_M_Inverter connection control"
                               Set_HWork_M := "Set_HWork_P3",
                               setPID_Pompy := "setPID_Pompy",
                               IsRunInverter_MA := "IsRunInverter_P1",
                               IsRunNetwork_MA := "IsRunNetwork_P1",
                               IsRunInverter_MB := "IsRunInverter_P2",
                               IsRunNetwork_MB := "IsRunNetwork_P2",
                               IsRunNetwork_MC := "IsRunNetwork_P3",
                               IsRunInverter_MC := "IsRunInverter_P3",
                               IsRunNetwork_MD := "IsRunInverter_P4",
                               IsRunInverter_MD := "IsRunInverter_P4",
                               FC2_Set_50H := "FC2_Set_50Hz",
                               IsRunInverter1 := "IsRunInverter1",
                               AlwaysTRUE := "AlwaysTRUE",
                               IsReady_MA := "IsReady_P1" AND "bitH_Aut_Man_P1",
                               IsReady_MB := "IsReady_P2" AND "bitH_Aut_Man_P2",
                               IsReady_MC := "IsReady_P3" AND "bitH_Aut_Man_P3",
                               IsReady_MD := "IsReady_P4" AND "bitH_Aut_Man_P4",
                               IsModeAut := "IsModeAut" AND "bitH_Aut_Man_P3",
                               FB9_Set_Motor2 := "FB9_Set_Motor2",
                               FB9_Set_Motor3 := "FB9_Set_Motor3",
                               FB9_Set_Motor4 := "FB9_Set_Motor4",
                               IsReady_Inverter := "IsReady_Inverter",
                               ResWorkInverter_to_MaxTime := "AlwaysFALSE",
                               number_pump := 3,
                               ActivePump := "dbdane".chosenPump,
                               setCMD_FM := "setCMD_FP3",
                               Timer_OFF_Inverter_M := "dbTimersForDrivers".Timer_OFF_Inverter_P3,
                               Timer_Start_Inver_M := "dbTimersForDrivers".Timer_Start_Inver_P3,
                               Timer_Set50Hz_Off_Inver_M := "dbTimersForDrivers".Timer_Hiteresis_On_Set50Hz_Inver_P3,
                               Mem_Res_setCMD_MC := "dbtags_Sterowanie".SetupControlPompownia.Mem_Res_setCMD_MC_P3,
                               setSUPV_FM => "setSUPV_FP3");
   END_IF;
END_REGION

